# B&R Automation Studio project ACOPOStrak_DATech_Pilot (part 5)

#### actCodeReader.st
```iecst
ACTION actCodeReader:

	IF gSim THEN

		gInitialDone := TRUE;

	END_IF

	IF NOT gInitialDone THEN

	CASE CodeStep OF

		CODE_WAIT:

			IF gShuttleTotalCount > checkSHCount THEN

					fbTrig.Enable				:= TRUE;

				IF fbTrig.Valid THEN

					CodeStep				:= CODE_CHECK_TRIG;

				END_IF

			ELSE

				gInitialDone				:= TRUE;
				fbTrig.Enable				:= FALSE;
//				gBarCodeReader.Enable 		:= FALSE;

			END_IF

		CODE_CHECK_TRIG:

			IF fbTrig.EventCount > 0 THEN

				checkSHCount := checkSHCount + 1;

				fbTrigInfo.Execute := TRUE;

				fbUserData.DataAddress 			:= ADR(userData);
				fbUserData.DataSize 			:= SIZE_OF_USERDATA;
				fbUserData.Mode					:= mcACPTRAK_USERDATA_GET;
				fbUserData.Execute 				:= TRUE;

				CodeStep						:= CODE_GET_SH;

			END_IF

		CODE_GET_SH:

			IF fbTrigInfo.Done = TRUE AND fbUserData.Done = TRUE THEN

				Axis	:= fbTrigInfo.TrgPointInfo.Axis;
				fbUserData.Execute 				:= FALSE;

				CodeStep 				:= CODE_MOVE_TO_READER;

			END_IF

		CODE_MOVE_TO_READER:

			fbMovelAbs.Sector				:= ADR(SectorTrackAll);
			fbMovelAbs.Axis 				:= ADR(Axis);

			fbMovelAbs.Velocity				:= gPar.MovementPar.Initialize.Velocity;
			fbMovelAbs.Acceleration 		:= gPar.MovementPar.Initialize.Acceleration;
			fbMovelAbs.Deceleration 		:= gPar.MovementPar.Initialize.Deceleration;
			fbMovelAbs.Position				:= POS_VISION;

			fbMovelAbs.Execute 				:= TRUE;

			fbMovelAbs.AdvancedParameters.StartDirection 		:= mcDIR_UNDEFINED;
			fbMovelAbs.AdvancedParameters.EndDirection 			:= mcDIR_POSITIVE;

			fbMovelAbs.AdvancedParameters.ShuttleOrientation 	:= mcDIR_UNDEFINED;
			fbMovelAbs.AdvancedParameters.PosRelativeTo 		:= mcACPTRAK_SEC_START;

			IF fbMovelAbs.Done THEN

				fbMovelAbs.Execute 			:= FALSE;

				CodeStep					:= CODE_READER_CHECK;

			END_IF

		CODE_READER_CHECK:

			IF gVisionSensor.DAT.StatusText = 'Ready' AND NOT gVisionSensor.DAT.ImageProcessingActive THEN

				gBarCodeReader.Trigger		:= TRUE;
				checkTakeCount				:= gBarCodeReader.TakeCount;
				CodeStep					:= CODE_CHECK_TAKE_COUNT;

			END_IF

		CODE_CHECK_TAKE_COUNT:

			IF gVisionSensor.DAT.ImageProcessingActive AND checkTakeCount <> gBarCodeReader.TakeCount THEN // gVisionSensor.DAT.StatusText <> 'Ready' AND checkTakeCount <> gBarCodeReader.TakeCount THEN //bNextStep1 THEN

				gBarCodeReader.Trigger		:= FALSE;

				CodeStep					:= CODE_ID_DEFINE;

			END_IF

		CODE_ID_DEFINE:

			IF NOT gVisionSensor.DAT.ImageProcessingActive THEN // bNextStep2 THEN //

//				fbUserData.Axis 		:= ADR(Axis);
				fbUserData.Mode 		:= mcACPTRAK_USERDATA_SET;
				fbUserData.Execute 		:= TRUE;
				fbUserData.DataAddress	:= ADR(userData);
				fbUserData.DataSize		:= SIZEOF(userData);

//				StrShuttleCount 		:= USINT_TO_STRING(checkSHCount);
//
//				IF checkSHCount < 10 THEN
//					userData.SerialNumber		:= 'FA99999900';
//					userData.SerialNumber		:= CONCAT(userData.SerialNumber, StrShuttleCount);
//
//				ELSIF checkSHCount < 100 THEN
//					userData.SerialNumber		:= 'FA9999990';
//					userData.SerialNumber		:= CONCAT(userData.SerialNumber, StrShuttleCount);
//				END_IF

//				brsmemcpy(ADR(userData.SerialNumber), ADR(StrTempShuttleID), 11);// ADR(gBarCodeReader.SerialNumber), 11);

				userData.SerialNumber := gBarCodeReader.SerialNumber;

				IF fbUserData.Done = TRUE THEN // AND bNextStep3 THEN

					fbUserData.Execute 	:= FALSE;
					CodeStep					:= CODE_RELEASE_SH;

				END_IF

			END_IF

		CODE_RELEASE_SH:

			fbMovelVel.Sector				:= ADR(SectorTrackAll);
			fbMovelVel.Axis 				:= ADR(Axis);

			fbMovelVel.RouteVelocity 		:= gPar.MovementPar.Initialize.RoutedVelocity;
			fbMovelVel.Velocity 			:= gPar.MovementPar.Initialize.Velocity;
			fbMovelVel.Acceleration 		:= gPar.MovementPar.Initialize.Acceleration;
			fbMovelVel.Deceleration 		:= gPar.MovementPar.Initialize.Deceleration;

			fbMovelVel.Execute 				:= TRUE;

			fbMovelVel.AdvancedParameters.StartDirection 		:= mcDIR_UNDEFINED;
			fbMovelVel.AdvancedParameters.EndDirection 			:= mcDIR_POSITIVE;

			fbMovelVel.AdvancedParameters.ShuttleOrientation 	:= mcDIR_UNDEFINED;
			fbMovelVel.AdvancedParameters.PosRelativeTo 		:= mcACPTRAK_SEC_START;

			CodeStep 					:= CODE_NORMAL_END;

//			IF fbMovelVel.Active THEN
//
//				fbMovelVel.Execute 			:= FALSE;
//				fbUserData.Execute			:= FALSE;
//				fbTrigInfo.Execute			:= FALSE;
//
//			END_IF

		CODE_NORMAL_END:

			fbTrigInfo.Execute			:= FALSE;
			fbUserData.Execute			:= FALSE;
			fbMovelVel.Execute 			:= FALSE;

			CodeStep 					:= CODE_WAIT;

		END_CASE

	END_IF

	fbTrig();
	fbTrigInfo();
	fbUserData();
	fbMovelAbs();
	fbMovelVel();
	ShReadInfo();

	bMoveVelActive 	:= fbMovelVel.Active;

END_ACTION

ACTION actCodeReader_INIT:

	CodeStep 			:= CODE_WAIT;

//	gBarCodeReader.Enable 		:= FALSE;
//	gBarCodeReader.Trigger		:= FALSE;

	checkSHCount		:= 0;

	fbTrig.Enable		:= FALSE;
	fbTrigInfo.Execute	:= FALSE;
	fbUserData.Execute	:= FALSE;
	fbMovelAbs.Execute	:= FALSE;
	fbMovelVel.Execute	:= FALSE;

END_ACTION

/////////////////////////////////////////////////////////////////////////////////////////////////////////

//
//		INIT_BARRIERSETTING:(* Process Point Setting *)
//			countShuttle					:= 0;
//			gShuttleTotalCount				:= 0;
//
//			fbCheckInStatus.Enable 			:= TRUE;
//
//			fbCheckIn.Command 				:= mcACPTRAK_BARRIER_CLOSE;
//			fbCheckIn.Execute 				:= TRUE;
//
//			fbCheckOut.Command 				:= mcACPTRAK_BARRIER_OPEN;
//			fbCheckOut.Execute 				:= TRUE;
//
//			IF fbCheckIn.Done = TRUE AND fbCheckOut.Done = TRUE	AND fbCheckInStatus.Valid = TRUE THEN
//				fbCheckIn.Execute 			:= FALSE;
//				fbCheckOut.Execute 			:= FALSE;
//
//				fbAsmGetShuttle.Assembly 		:= ADR(gAsmMain);
//				fbAsmGetShuttle.Enable 			:= TRUE;
//
//				IF fbAsmGetShuttle.Valid = TRUE THEN
//					gShuttleTotalCount			:= fbAsmGetShuttle.TotalCount;
//					initStep 					:= INIT_SHUTTLE_CHECK;
//				END_IF
//			END_IF
//
//		INIT_SHUTTLE_CHECK:
//			IF fbAsmGetShuttle.TotalCount > countShuttle THEN
//				readShuttleInfo.Axis  		:= ADR(fbAsmGetShuttle.Axis);
//				readShuttleInfo.Enable 		:= TRUE;
//
//				IF readShuttleInfo.Valid = TRUE THEN
//					countShuttle			:= countShuttle + 1;
//					fbAsmGetShuttle.Next	:= FALSE;
//					initStep 				:= INIT_MOVE;
//				END_IF
//			ELSE
//				fbAsmGetShuttle.Enable 		:= FALSE;
//				readShuttleInfo.Enable 		:= FALSE;
//				initStep 					:= INIT_ADD_TICKET;
//			END_IF
//
//		INIT_MOVE:
//			IF readShuttleInfo.ShuttleInfo.CurrentValues.Velocity = 0 THEN
//				fbMovelVel.Sector				:= ADR(SecMain);
//				fbMovelVel.Axis 				:= ADR(fbAsmGetShuttle.Axis);
//
//				fbMovelVel.RouteVelocity 		:= gPar.MovementPar.Initialize.RoutedVelocity;
//				fbMovelVel.Velocity 			:= gPar.MovementPar.Initialize.Velocity;
//				fbMovelVel.Acceleration 		:= gPar.MovementPar.Initialize.Acceleration;
//				fbMovelVel.Deceleration 		:= gPar.MovementPar.Initialize.Deceleration;
//				fbMovelVel.Execute 				:= TRUE;
//
//				fbMovelVel.AdvancedParameters.StartDirection 		:= mcDIR_UNDEFINED;
//				fbMovelVel.AdvancedParameters.EndDirection 			:= mcDIR_POSITIVE;
//
//				fbMovelVel.AdvancedParameters.ShuttleOrientation 	:= mcDIR_UNDEFINED;
//				fbMovelVel.AdvancedParameters.PosRelativeTo 		:= mcACPTRAK_SEC_START;
//
//				IF bMoveVelActive = FALSE AND fbMovelVel.Active = TRUE THEN
//					fbMovelVel.Execute 			:= FALSE;
//					readShuttleInfo.Enable 		:= FALSE;
//					fbAsmGetShuttle.Next		:= TRUE;
//					initStep 					:= INIT_SHUTTLE_CHECK;
//				END_IF
//			END_IF
//
//		INIT_ADD_TICKET:
//			fbCheckIn.AdvancedParameters.TicketCount 	:= gShuttleTotalCount;
//			fbCheckIn.Command							:= mcACPTRAK_BARRIER_ADD_TICKETS;
//			fbCheckIn.Execute 							:= TRUE;
//
//			IF fbCheckIn.Done = TRUE THEN
//				fbCheckIn.Execute						:= FALSE;
//				initStep 								:= INIT_START_ID_IDENTIFICATION;
//			END_IF
//
//
//		INIT_START_ID_IDENTIFICATION:
//			IF fbCheckInStatus.BarrierInfo.RemainingTickets = 0 THEN
//				initStep 								:= INIT_CHECK_END;
//			END_IF
//
//		INIT_CHECK_END:
//			fbSecGetShuttles.Sector := ADR(SecMain);
//			fbSecGetShuttles.Enable := TRUE;
//			fbSecGetShuttles.AdvancedParameters.StartPosition 	:= 1.2;
//			fbSecGetShuttles.AdvancedParameters.EndPosition 	:= 2.4;
//
//			IF fbSecGetShuttles.Valid = TRUE THEN
//				IF fbSecGetShuttles.TotalCount = 0 THEN
//					fbSecGetShuttles.Enable 			:= FALSE;
//					initStep 							:= INIT_NORMAL_END;
//				ELSE
//					fbSecGetShuttles.Enable := FALSE;
//				END_IF
//			END_IF
//
//		INIT_NORMAL_END:
//			fbCheckInStatus.Enable := FALSE;
//			fbCheckIn.Execute := TRUE;
//			fbCheckOut.Execute := TRUE;
//
//			fbCheckIn.Command := mcACPTRAK_BARRIER_OPEN;
//			fbCheckOut.Command := mcACPTRAK_BARRIER_OPEN;
//
//			IF fbCheckIn.Done = TRUE AND fbCheckOut.Done = TRUE THEN
//				gSts.AsmState 					:= E_ASM_IDLE;
//			END_IF
//	END_CASE;
//
//	fbCheckInStatus();
//	fbCheckIn();
//	fbCheckOut();
//
//	fbAsmGetShuttle();
//	readShuttleInfo();
//
//	fbSecGetShuttles();
//
//	bMoveVelActive 	:= fbMovelVel.Active;
//
//END_ACTION
//
//ACTION actInitialize_INIT:
//	CodeStep 						:= CODE_WAIT;
//	fbAsmGetShuttle.Enable 			:= FALSE;
//	fbSecGetShuttles.Enable 		:= FALSE;
//	fbCheckInStatus.Enable			:= FALSE;
//	fbCheckIn.Execute 				:= FALSE;
//	fbCheckOut.Execute 				:= FALSE;
//	fbMovelVel.Execute				:= FALSE;
//END_ACTION
```

### Program Logical/Source/AsmControl/ctrCleanMode (IEC)

#### Variables.var
```iecst
VAR
	initStep : INT;
END_VAR
(**)
VAR
	fbSecGetShuttles : MC_BR_SecGetShuttleSel_AcpTrak;
END_VAR
(**)
VAR
	fbMovelVel : MC_BR_RoutedMoveVel_AcpTrak;
	fbMoveAbs : MC_BR_RoutedMoveAbs_AcpTrak;
END_VAR
(**)
VAR
	bMoveVelActive : BOOL;
END_VAR
(**)
VAR
	fbCheckOutStatus : MC_BR_BarrierReadInfo_AcpTrak;
	fbCheckInStatus : MC_BR_BarrierReadInfo_AcpTrak;
	fbCheckIn : MC_BR_BarrierCommand_AcpTrak;
	fbCheckOut : MC_BR_BarrierCommand_AcpTrak;
	fbCheckInTrg : MC_BR_TrgPointEnable_AcpTrak;
	fbCheckInTrgInfo : MC_BR_TrgPointGetInfo_AcpTrak;
	TotalShuttleCount : DINT;
END_VAR
```

#### Main.st
```iecst
PROGRAM _INIT

	fbCheckIn.ProcessPoint			:= ADR(ptCheckIn);
	fbCheckInStatus.ProcessPoint 	:= ADR(ptCheckIn);
	fbCheckInTrg.ProcessPoint		:= ADR(ptCheckIn);
	fbCheckInTrgInfo.ProcessPoint	:= ADR(ptCheckIn);

	fbCheckOutStatus.ProcessPoint	:= ADR(ptCheckOut);
	fbCheckOut.ProcessPoint			:= ADR(ptCheckOut);

END_PROGRAM

PROGRAM _CYCLIC

	IF gSts.AsmState <> E_ASM_CLEAN THEN
		initStep					:= 0;

		fbSecGetShuttles.Enable		:= FALSE;
		fbCheckInTrgInfo.Execute	:= FALSE;
		fbCheckIn.Execute			:= FALSE;
		fbCheckInStatus.Enable		:= FALSE;

		fbMoveAbs.Execute				:= FALSE;
		fbMovelVel.Execute 				:= FALSE;

		TotalShuttleCount				:= 0;
	ELSE

		CASE initStep OF
			0:
				fbCheckInStatus.Enable	:= TRUE;
				fbCheckIn.Execute 		:= TRUE;
				fbCheckOut.Execute 		:= TRUE;

				fbCheckIn.Command 		:= mcACPTRAK_BARRIER_OPEN;
				fbCheckOut.Command 		:= mcACPTRAK_BARRIER_OPEN;

				IF fbCheckIn.Done AND fbCheckInStatus.Valid THEN
					fbCheckIn.Execute 	:= FALSE;
					fbCheckOut.Execute 	:= FALSE;
					initStep			:= 10;
				END_IF

			10:
				fbSecGetShuttles.Sector := ADR(SectorTrackAll);
				fbSecGetShuttles.Enable := TRUE;
				fbSecGetShuttles.AdvancedParameters.StartPosition	:= 0.0;
				fbSecGetShuttles.AdvancedParameters.EndPosition		:= 0.0;

				IF fbSecGetShuttles.Valid = TRUE THEN
					TotalShuttleCount 	:= fbSecGetShuttles.TotalCount;
					initStep 			:= 20;
				END_IF

			20:
				fbSecGetShuttles.Next 			:= FALSE;

				fbMovelVel.Sector				:= ADR(SectorTrackAll);
				fbMovelVel.Axis 				:= ADR(fbSecGetShuttles.Axis);

				fbMovelVel.Position				:= 12.48;
				fbMovelVel.RouteVelocity 		:= 1.0;
				fbMovelVel.Velocity 			:= 1.0;
				fbMovelVel.Acceleration 		:= 1.0;
				fbMovelVel.Deceleration 		:= 1.0;
				fbMovelVel.Execute 				:= TRUE;

				fbMovelVel.AdvancedParameters.StartDirection 		:= mcDIR_POSITIVE;
				fbMovelVel.AdvancedParameters.EndDirection 			:= mcDIR_UNDEFINED;
				fbMovelVel.AdvancedParameters.ShuttleOrientation 	:= mcDIR_UNDEFINED;

				IF bMoveVelActive = FALSE AND fbMovelVel.Active = TRUE THEN
					fbMovelVel.Execute 			:= FALSE;
					initStep 					:= 30;
				END_IF

			30:
				IF fbSecGetShuttles.RemainingCount > 0 THEN
					fbSecGetShuttles.Next 		:= TRUE;
					initStep 					:= 20;
				ELSE
					fbSecGetShuttles.Enable 	:= FALSE;
			//		initStep 					:= 40;
				END_IF

			40:
				IF fbCheckInStatus.BarrierInfo.RemainingTickets = 0 THEN
					initStep 					:= 50;
				END_IF

			50:
				fbSecGetShuttles.Sector 		:= ADR(SectorTrackAll);
				fbSecGetShuttles.Enable 		:= TRUE;
				fbSecGetShuttles.AdvancedParameters.StartPosition 	:= 13.14;//12.48; // Check in point
				fbSecGetShuttles.AdvancedParameters.EndPosition 	:= 0.0;

				IF fbSecGetShuttles.Valid = TRUE AND fbSecGetShuttles.TotalCount = 0 THEN
					fbSecGetShuttles.Enable 		:= FALSE;
					initStep 						:= 60;
				ELSIF  fbSecGetShuttles.Valid = TRUE AND fbSecGetShuttles.TotalCount > 0 THEN
					fbSecGetShuttles.Enable 		:= FALSE;
				END_IF

			60:
				fbCheckInStatus.Enable := FALSE;
				fbCheckIn.Execute := TRUE;
				fbCheckOut.Execute := TRUE;

				fbCheckIn.Command := mcACPTRAK_BARRIER_OPEN;
				fbCheckOut.Command := mcACPTRAK_BARRIER_OPEN;

				IF fbCheckIn.Done = TRUE AND fbCheckOut.Done = TRUE THEN
					fbCheckIn.Execute 			:= FALSE;
					fbCheckOut.Execute 			:= FALSE;
					fbSecGetShuttles.Enable 	:= FALSE;
					gSts.AsmState 				:= E_ASM_IDLE;
					initStep 					:= 0;
				END_IF

		END_CASE;
	END_IF

	fbSecGetShuttles();

	fbCheckInTrg();
	fbCheckInTrgInfo();
	fbCheckIn();
	fbCheckInStatus();
	fbCheckOut();
	fbCheckOutStatus();
//	fbUserData();

	fbMoveAbs();
	bMoveVelActive 	:= fbMovelVel.Active;
	fbMovelVel();

END_PROGRAM

PROGRAM _EXIT
	(* Insert code here *)

END_PROGRAM
```

### Program Logical/Source/Control/ctrTransfer (IEC)

#### Main.st - Init, cyclic, exit code
```iecst
PROGRAM _INIT

	gSim	:= DiagCpuIsSimulated();

	StStage[0].Sector		:= ADR(SectorCurve1);
	StStage[1].Sector		:= ADR(SectorTrackA_2);
	StStage[2].Sector		:= ADR(SectorTrackA_2);
	StStage[3].Sector		:= ADR(SectorTrackA_2);
	StStage[4].Sector		:= ADR(SectorTrackA_2);
	StStage[5].Sector		:= ADR(SectorTrackA_2);
	StStage[6].Sector		:= ADR(SectorTrackA_2);
	StStage[7].Sector		:= ADR(SectorTrackA_2);
	StStage[8].Sector		:= ADR(SectorTrackA_2);
	StStage[9].Sector		:= ADR(SectorTrackA_3);
	StStage[10].Sector		:= ADR(SectorCurve3);
	StStage[11].Sector		:= ADR(SectorTrackA_4);
	StStage[12].Sector		:= ADR(SectorTrackA_4);
	StStage[13].Sector		:= ADR(SectorTrackA_4);
	StStage[14].Sector		:= ADR(SectorTrackA_4);
	StStage[15].Sector		:= ADR(SectorTrackA_4);
	StStage[16].Sector		:= ADR(SectorCurve4);
	StStage[17].Sector		:= ADR(SectorCurve4);
	StStage[18].Sector		:= ADR(SectorTrackA_1);

	/////////////////////////////////////////////////////////////////////////////////////
	// Can supply
	fbStage1.CheckInProcessPoint		:= ADR(ptCheckIn);
	fbStage1.CheckOutProcessPoint		:= ADR(ptCheckOut);
	fbStage1.TargetStage				:= ADR(StStage[0]);
	fbStage1.TargetSlotCount			:= COUNT_OF_SLOT;
	// TC insert
	fbStage2.SourceStage[0]				:= ADR(StStage[0]);
	fbStage2.SourceSlotCount[0]			:= COUNT_OF_SLOT;
	fbStage2.TargetStage				:= ADR(StStage[1]);
	fbStage2.TargetSlotCount			:= COUNT_OF_SLOT;
	// TC push
	fbStage3.SourceStage[0]				:= ADR(StStage[1]);
	fbStage3.SourceSlotCount[0]			:= COUNT_OF_SLOT;
	fbStage3.TargetStage				:= ADR(StStage[2]);
	fbStage3.TargetSlotCount			:= COUNT_OF_SLOT;
	// TC vision
	fbStage4.SourceStage[0]				:= ADR(StStage[2]);
	fbStage4.SourceSlotCount[0]			:= COUNT_OF_SLOT;
	fbStage4.TargetStage				:= ADR(StStage[3]);
	fbStage4.TargetSlotCount			:= COUNT_OF_SLOT;
	// TC NG re-insert
	fbStage5.SourceStage[0]				:= ADR(StStage[3]);
	fbStage5.SourceSlotCount[0]			:= COUNT_OF_SLOT;
	fbStage5.TargetStage				:= ADR(StStage[4]);
	fbStage5.TargetSlotCount			:= COUNT_OF_SLOT;
	// BCR vision
	fbStage6.SourceStage[0]				:= ADR(StStage[4]);
	fbStage6.SourceSlotCount[0]			:= COUNT_OF_SLOT;
	fbStage6.TargetStage				:= ADR(StStage[5]);
	fbStage6.TargetSlotCount			:= COUNT_OF_SLOT;
	// CCR 1
	fbStage7.SourceStage[0]				:= ADR(StStage[5]);
	fbStage7.SourceSlotCount[0]			:= COUNT_OF_SLOT;
	fbStage7.TargetStage				:= ADR(StStage[6]);
	fbStage7.TargetSlotCount			:= COUNT_OF_SLOT;
	// CCR 1 vision
	fbStage8.SourceStage[0]				:= ADR(StStage[6]);
	fbStage8.SourceSlotCount[0]			:= COUNT_OF_SLOT;
	fbStage8.TargetStage				:= ADR(StStage[7]);
	fbStage8.TargetSlotCount			:= COUNT_OF_SLOT;
	// CCR 2
	fbStage9.SourceStage[0]				:= ADR(StStage[7]);
	fbStage9.SourceSlotCount[0]			:= COUNT_OF_SLOT;
	fbStage9.TargetStage				:= ADR(StStage[8]);
	fbStage9.TargetSlotCount			:= COUNT_OF_SLOT;
	// Maint
	fbStage10.SourceStage[0]			:= ADR(StStage[8]);
	fbStage10.SourceSlotCount[0]		:= COUNT_OF_SLOT;
	fbStage10.TargetStage				:= ADR(StStage[9]);
	fbStage10.TargetSlotCount			:= COUNT_OF_SLOT;
	// CCR 2 vision
	fbStage11.SourceStage[0]			:= ADR(StStage[9]);
	fbStage11.SourceSlotCount[0]		:= COUNT_OF_SLOT;
	fbStage11.TargetStage				:= ADR(StStage[10]);
	fbStage11.TargetSlotCount			:= COUNT_OF_SLOT;
	// CCR 3
	fbStage12.SourceStage[0]			:= ADR(StStage[10]);
	fbStage12.SourceSlotCount[0]		:= COUNT_OF_SLOT;
	fbStage12.TargetStage				:= ADR(StStage[11]);
	fbStage12.TargetSlotCount			:= COUNT_OF_SLOT;
	// CCR 3 vision
	fbStage13.SourceStage[0]			:= ADR(StStage[11]);
	fbStage13.SourceSlotCount[0]		:= COUNT_OF_SLOT;
	fbStage13.TargetStage				:= ADR(StStage[12]);
	fbStage13.TargetSlotCount			:= COUNT_OF_SLOT;
	// CSZ
	fbStage14.SourceStage[0]			:= ADR(StStage[12]);
	fbStage14.SourceSlotCount[0]		:= COUNT_OF_SLOT;
	fbStage14.TargetStage				:= ADR(StStage[13]);
	fbStage14.TargetSlotCount			:= COUNT_OF_SLOT;
	// 3D done position
	fbStage15.SourceStage[0]			:= ADR(StStage[13]);
	fbStage15.SourceSlotCount[0]		:= COUNT_OF_SLOT;
	fbStage15.TargetStage				:= ADR(StStage[14]);
	fbStage15.TargetSlotCount			:= COUNT_OF_SLOT;
	// Diameter inspection
	fbStage16.SourceStage[0]			:= ADR(StStage[14]);
	fbStage16.SourceSlotCount[0]		:= COUNT_OF_SLOT;
	fbStage16.TargetStage				:= ADR(StStage[15]);
	fbStage16.TargetSlotCount			:= COUNT_OF_SLOT;
	// NG out
	fbStage17.SourceStage[0]			:= ADR(StStage[15]);
	fbStage17.SourceSlotCount[0]		:= COUNT_OF_SLOT;
	fbStage17.TargetStage				:= ADR(StStage[16]);
	fbStage17.TargetSlotCount			:= COUNT_OF_SLOT;
	// Unloading
	fbStage18.SourceStage[0]			:= ADR(StStage[16]);
	fbStage18.SourceSlotCount[0]		:= COUNT_OF_SLOT;
	fbStage18.TargetStage				:= ADR(StStage[17]);
	fbStage18.TargetSlotCount			:= COUNT_OF_SLOT;
	// Clean
	fbStage19.SourceStage[0]			:= ADR(StStage[17]);
	fbStage19.SourceSlotCount[0]		:= COUNT_OF_SLOT;
	fbStage19.TargetStage				:= ADR(StStage[18]);
	fbStage19.TargetSlotCount			:= COUNT_OF_SLOT;
	// Return
	fbReturn.SourceStage[0]				:= ADR(StStage[18]);
	fbReturn.SourceSlotCount[0]			:= COUNT_OF_SLOT;
	fbReturn.TargetSector				:= ADR(SectorTrackAll);
	fbReturn.TargetPosition				:= 12.5;
	/////////////////////////////////////////////////////////////////////////////////////
	InitializeFcBank(30);

	actParameterInitialize;

	/////////////////////////////////////////////////////////////////////////////////////
	// Buffer
	/////////////////////////////////////////////////////////////////////////////////////

	//Wait buffer for CSZ
	fbCSZWait.InPoint				:= ADR(ptCSZIn);
	fbCSZWait.OutPoint				:= ADR(ptCSZOut);
	fbCSZWait.MaximumShuttleCount	:= 1;
	//fbCSZWait.InitShuttleCount		:= 1;

	//Wait for unloading
	fbUnloadingWait.InPoint				:= ADR(ptUnloadingIn);
	fbUnloadingWait.OutPoint			:= ADR(ptUnloadingOut);
	fbUnloadingWait.MaximumShuttleCount	:= 1;
	fbUnloadingWait.InitShuttleCount	:= 1;

END_PROGRAM

PROGRAM _CYCLIC

	actUpdateParamter;

	CASE gSts.AsmState OF
		E_ASM_INITIALIZATION:
			//For Initialize Slot Status.
			FOR i := 0 TO 18 DO
				StStage[i].Interface	:= E_SLOT_UNKNOWN;
			END_FOR;

		E_ASM_MANUAL:

			fbStage1(Enable := TRUE, Process := FALSE, Feeding := FALSE);
			fbStage2(Enable := TRUE, Process := FALSE);
			fbStage3(Enable := TRUE, Process := FALSE);
			fbStage4(Enable := TRUE, Process := FALSE);
			fbStage5(Enable := TRUE, Process := FALSE);
			fbStage6(Enable := TRUE, Process := FALSE);
			fbStage7(Enable := TRUE, Process := FALSE);
			fbStage8(Enable := TRUE, Process := FALSE);
			fbStage9(Enable := TRUE, Process := FALSE);
			fbStage10(Enable := TRUE, Process := FALSE);
			fbStage11(Enable := TRUE, Process := FALSE);
			fbStage12(Enable := TRUE, Process := FALSE);
			fbStage13(Enable := TRUE, Process := FALSE);
			fbStage14(Enable := TRUE, Process := FALSE);
			fbStage15(Enable := TRUE, Process := FALSE);
			fbStage16(Enable := TRUE, Process := FALSE);
			fbStage17(Enable := TRUE, Process := FALSE);
			fbStage18(Enable := TRUE, Process := FALSE);
			fbStage19(Enable := TRUE, Process := FALSE);
			fbReturn(Enable := TRUE, Process := FALSE);
			fbCSZWait(Enable := FALSE);
			fbUnloadingWait(Enable := FALSE);

			FOR i := 0 TO 18 DO
				StStage[i].Interface	:= E_SLOT_MANUAL;

				IF i < 18 THEN
					StStage[i].NextStage	:= ADR(StStage[i + 1]);
				ELSIF i = 18 THEN
					StStage[18].NextStage	:= ADR(StStage[0]);
				END_IF
			END_FOR;

		E_ASM_IDLE:

			fbStage1(Enable := TRUE, Process := TRUE, Feeding := FALSE);
			fbStage2(Enable := TRUE, Process := TRUE);
			fbStage3(Enable := TRUE, Process := TRUE);
			fbStage4(Enable := TRUE, Process := TRUE);
			fbStage5(Enable := TRUE, Process := TRUE);
			fbStage6(Enable := TRUE, Process := TRUE);
			fbStage7(Enable := TRUE, Process := TRUE);
			fbStage8(Enable := TRUE, Process := TRUE);
			fbStage9(Enable := TRUE, Process := TRUE);
			fbStage10(Enable := TRUE, Process := TRUE);
			fbStage11(Enable := TRUE, Process := TRUE);
			fbStage12(Enable := TRUE, Process := TRUE);
			fbStage13(Enable := TRUE, Process := TRUE);
			fbStage14(Enable := TRUE, Process := TRUE);
			fbStage15(Enable := TRUE, Process := TRUE);
			fbStage16(Enable := TRUE, Process := TRUE);
			fbStage17(Enable := TRUE, Process := TRUE);
			fbStage18(Enable := TRUE, Process := TRUE);
			fbStage19(Enable := TRUE, Process := TRUE);
			fbReturn(Enable := TRUE, Process := TRUE);
			fbCSZWait(Enable := TRUE);
			fbUnloadingWait(Enable := TRUE);

		E_ASM_PROCESS:

			fbStage1(Enable := TRUE, Process := TRUE, Feeding := TRUE);
			fbStage2(Enable := TRUE, Process := TRUE);
			fbStage3(Enable := TRUE, Process := TRUE);
			fbStage4(Enable := TRUE, Process := TRUE);
			fbStage5(Enable := TRUE, Process := TRUE);
			fbStage6(Enable := TRUE, Process := TRUE);
			fbStage7(Enable := TRUE, Process := TRUE);
			fbStage8(Enable := TRUE, Process := TRUE);
			fbStage9(Enable := TRUE, Process := TRUE);
			fbStage10(Enable := TRUE, Process := TRUE);
			fbStage11(Enable := TRUE, Process := TRUE);
			fbStage12(Enable := TRUE, Process := TRUE);
			fbStage13(Enable := TRUE, Process := TRUE);
			fbStage14(Enable := TRUE, Process := TRUE);
			fbStage15(Enable := TRUE, Process := TRUE);
			fbStage16(Enable := TRUE, Process := TRUE);
			fbStage17(Enable := TRUE, Process := TRUE);
			fbStage18(Enable := TRUE, Process := TRUE);
			fbStage19(Enable := TRUE, Process := TRUE);
			fbReturn(Enable := TRUE, Process := TRUE);
			fbCSZWait(Enable := TRUE);
			fbUnloadingWait(Enable := TRUE);

		E_ASM_STOPPING:

			fbStage1(Enable := TRUE, Process := TRUE, Feeding := FALSE);
			fbStage2(Enable := TRUE, Process := TRUE);
			fbStage3(Enable := TRUE, Process := TRUE);
			fbStage4(Enable := TRUE, Process := TRUE);
			fbStage5(Enable := TRUE, Process := TRUE);
			fbStage6(Enable := TRUE, Process := TRUE);
			fbStage7(Enable := TRUE, Process := TRUE);
			fbStage8(Enable := TRUE, Process := TRUE);
			fbStage9(Enable := TRUE, Process := TRUE);
			fbStage10(Enable := TRUE, Process := TRUE);
			fbStage11(Enable := TRUE, Process := TRUE);
			fbStage12(Enable := TRUE, Process := TRUE);
			fbStage13(Enable := TRUE, Process := TRUE);
			fbStage14(Enable := TRUE, Process := TRUE);
			fbStage15(Enable := TRUE, Process := TRUE);
			fbStage16(Enable := TRUE, Process := TRUE);
			fbStage17(Enable := TRUE, Process := TRUE);
			fbStage18(Enable := TRUE, Process := TRUE);
			fbStage19(Enable := TRUE, Process := TRUE);
			fbReturn(Enable := TRUE, Process := TRUE);
			fbCSZWait(Enable := TRUE);
			fbUnloadingWait(Enable := TRUE);

			IF fbStage1.ErrorID = MyTrakIdle AND
				fbStage2.ErrorID = MyTrakIdle AND
				fbStage3.ErrorID = MyTrakIdle AND
				fbStage4.ErrorID = MyTrakIdle AND
				fbStage5.ErrorID = MyTrakIdle AND
				fbStage6.ErrorID = MyTrakIdle AND
				fbStage7.ErrorID = MyTrakIdle AND
				fbStage8.ErrorID = MyTrakIdle AND
				fbStage9.ErrorID = MyTrakIdle AND
				fbStage10.ErrorID = MyTrakIdle AND
				fbStage11.ErrorID = MyTrakIdle AND
				fbStage12.ErrorID = MyTrakIdle AND
				fbStage13.ErrorID = MyTrakIdle AND
				fbStage14.ErrorID = MyTrakIdle AND
				fbStage15.ErrorID = MyTrakIdle AND
				fbStage16.ErrorID = MyTrakIdle AND
				fbStage17.ErrorID = MyTrakIdle AND
				fbStage18.ErrorID = MyTrakIdle AND
				fbStage19.ErrorID = MyTrakIdle AND

				StStage[0].Interface = E_SLOT_IDLE AND
				StStage[1].Interface = E_SLOT_IDLE AND
				StStage[2].Interface = E_SLOT_IDLE AND
				StStage[3].Interface = E_SLOT_IDLE AND
				StStage[4].Interface = E_SLOT_IDLE AND
				StStage[5].Interface = E_SLOT_IDLE AND
				StStage[6].Interface = E_SLOT_IDLE AND
				StStage[7].Interface = E_SLOT_IDLE AND
				StStage[8].Interface = E_SLOT_IDLE AND
				StStage[9].Interface = E_SLOT_IDLE AND
				StStage[10].Interface = E_SLOT_IDLE AND
				StStage[11].Interface = E_SLOT_IDLE AND
				StStage[12].Interface = E_SLOT_IDLE AND
				StStage[13].Interface = E_SLOT_IDLE AND
				StStage[14].Interface = E_SLOT_IDLE AND
				StStage[15].Interface = E_SLOT_IDLE AND
				StStage[16].Interface = E_SLOT_IDLE AND
				StStage[17].Interface = E_SLOT_IDLE AND
				StStage[18].Interface = E_SLOT_IDLE	THEN
			//	gSts.AsmState	:= E_ASM_IDLE;
			END_IF

		ELSE
			fbStage1(Enable := FALSE, Process := FALSE, Feeding := FALSE);
			fbStage2(Enable := FALSE, Process := FALSE);
			fbStage3(Enable := FALSE, Process := FALSE);
			fbStage4(Enable := FALSE, Process := FALSE);
			fbStage5(Enable := FALSE, Process := FALSE);
			fbStage6(Enable := FALSE, Process := FALSE);
			fbStage7(Enable := FALSE, Process := FALSE);
			fbStage8(Enable := FALSE, Process := FALSE);
			fbStage9(Enable := FALSE, Process := FALSE);
			fbStage10(Enable := FALSE, Process := FALSE);
			fbStage11(Enable := FALSE, Process := FALSE);
			fbStage12(Enable := FALSE, Process := FALSE);
			fbStage13(Enable := FALSE, Process := FALSE);
			fbStage14(Enable := FALSE, Process := FALSE);
			fbStage15(Enable := FALSE, Process := FALSE);
			fbStage16(Enable := FALSE, Process := FALSE);
			fbStage17(Enable := FALSE, Process := FALSE);
			fbStage18(Enable := FALSE, Process := FALSE);
			fbStage19(Enable := FALSE, Process := FALSE);
			fbReturn(Enable := FALSE, Process := FALSE);
			fbCSZWait(Enable := FALSE);
			fbUnloadingWait(Enable := FALSE);

	END_CASE;

	readShuttleInfo.Axis	:= ADR(StStage[0].Shuttle);
	readShuttleInfo();

END_PROGRAM

PROGRAM _EXIT

	fbStage1.Enable		:= FALSE;
	fbStage2.Enable		:= FALSE;
	fbStage3.Enable		:= FALSE;
	fbStage4.Enable		:= FALSE;
	fbStage5.Enable		:= FALSE;
	fbStage6.Enable		:= FALSE;
	fbStage7.Enable		:= FALSE;
	fbStage8.Enable		:= FALSE;
	fbStage9.Enable		:= FALSE;
	fbStage10.Enable	:= FALSE;
	fbStage11.Enable	:= FALSE;
	fbStage12.Enable	:= FALSE;
	fbStage13.Enable	:= FALSE;
	fbStage14.Enable	:= FALSE;
	fbStage15.Enable	:= FALSE;
	fbStage16.Enable	:= FALSE;
	fbStage17.Enable	:= FALSE;
	fbStage18.Enable	:= FALSE;
	fbStage19.Enable	:= FALSE;
	fbCSZWait.Enable	:= FALSE;

END_PROGRAM
```

#### Variables.var - Local variables
```iecst
VAR
	fbStage1 : MyTrak_Buffer; (*can supply*)
	fbStage2 : MyTrak_TransStage; (*TC insert*)
	fbStage3 : MyTrak_TransStage; (*TC push*)
	fbStage4 : MyTrak_TransStage; (*TC vision*)
	fbStage5 : MyTrak_TransStage; (*TC NG re-insert*)
	fbStage6 : MyTrak_TransStage; (*BCR vision*)
	fbStage7 : MyTrak_TransStage; (*CCR 1*)
	fbStage8 : MyTrak_TransStage; (*CCR 1 vision*)
	fbStage9 : MyTrak_TransStage; (*CCR 2 *)
	fbStage10 : MyTrak_TransStage; (*Maint*)
	fbStage11 : MyTrak_TransStage; (*CCR 2 vision*)
	fbStage12 : MyTrak_TransStage; (*CCR 3*)
	fbStage13 : MyTrak_TransStage; (*CCR 3 vision*)
	fbStage14 : MyTrak_TransStage; (*CSZ*)
	fbStage15 : MyTrak_TransStage; (*3D scan done position*)
	fbStage16 : MyTrak_TransStage; (*Diameter inspection*)
	fbStage17 : MyTrak_TransStage; (*NG out*)
	fbStage18 : MyTrak_TransStage; (*unloading*)
	fbStage19 : MyTrak_TransStage; (*Clean*)
	fbReturn : MyTrak_Serialize;
	fbCSZWait : MyTrak_TicketArea;
	fbUnloadingWait : MyTrak_TicketArea;
END_VAR
(**)
VAR
	readShuttleInfo : MC_BR_ShReadInfo_AcpTrak;
	i : USINT;
END_VAR
```

#### actUpdateParameter.st
```iecst
ACTION actUpdateParamter:

	// Stage pararmeter setting
	FOR i := 0 TO 18 DO
		StStage[i].Enable	:= TRUE;
	END_FOR;

	StStage[0].Position			:= POS_STAGE1 + gPar.PositionOffset.Stage[0];
	StStage[1].Position			:= POS_STAGE2 + gPar.PositionOffset.Stage[1];
	StStage[2].Position			:= POS_STAGE3 + gPar.PositionOffset.Stage[2];
	StStage[3].Position			:= POS_STAGE4 + gPar.PositionOffset.Stage[3];
	StStage[4].Position			:= POS_STAGE5 + gPar.PositionOffset.Stage[4];
	StStage[5].Position			:= POS_STAGE6 + gPar.PositionOffset.Stage[5];
	StStage[6].Position			:= POS_STAGE7 + gPar.PositionOffset.Stage[6];
	StStage[7].Position			:= POS_STAGE8 + gPar.PositionOffset.Stage[7];
	StStage[8].Position			:= POS_STAGE9 + gPar.PositionOffset.Stage[8];
	StStage[9].Position			:= POS_STAGE10 + gPar.PositionOffset.Stage[9];
	StStage[10].Position		:= POS_STAGE11 + gPar.PositionOffset.Stage[10];
	StStage[11].Position		:= POS_STAGE12 + gPar.PositionOffset.Stage[11];
	StStage[12].Position		:= POS_STAGE13 + gPar.PositionOffset.Stage[12];
	StStage[13].Position		:= POS_STAGE14 + gPar.PositionOffset.Stage[13];
	StStage[14].Position		:= POS_STAGE15 + gPar.PositionOffset.Stage[14];
	StStage[15].Position		:= POS_STAGE16 + gPar.PositionOffset.Stage[15];
	StStage[16].Position		:= POS_STAGE17 + gPar.PositionOffset.Stage[16];
	StStage[17].Position		:= POS_STAGE18 + gPar.PositionOffset.Stage[17];
	StStage[18].Position		:= POS_STAGE19 + gPar.PositionOffset.Stage[18];

	// Movement pararmeter setting

	fbStage1.SetPPM										:= gPar.TargetPPM;
	fbStage1.CountOfOneShot								:= gPar.CountOfGroup;
	fbStage1.Velocity									:= gPar.MovementPar.Stage1.Velocity;
	fbStage1.Acceleration								:= gPar.MovementPar.Stage1.Acceleration;
	fbStage1.Deceleration								:= gPar.MovementPar.Stage1.Deceleration;
	fbStage1.AdvancedParameters.StartDirection 			:= mcDIR_POSITIVE;
	fbStage1.AdvancedParameters.EndDirection 			:= mcDIR_UNDEFINED;
	fbStage1.AdvancedParameters.ShuttleOrientation 		:= mcDIR_UNDEFINED;
	fbStage1.MaximumShuttleCount						:= gPar.MovementPar.Stage1.MaxController;

	fbStage2.Velocity									:= gPar.MovementPar.Stage2.Velocity;
	fbStage2.Acceleration								:= gPar.MovementPar.Stage2.Acceleration;
	fbStage2.Deceleration								:= gPar.MovementPar.Stage2.Deceleration;
	fbStage2.AdvancedParameters.StartDirection 			:= mcDIR_POSITIVE;
	fbStage2.AdvancedParameters.EndDirection 			:= mcDIR_UNDEFINED;
	fbStage2.AdvancedParameters.ShuttleOrientation 		:= mcDIR_UNDEFINED;
	fbStage2.MaximumShuttleCount						:= gPar.MovementPar.Stage2.MaxController;

	fbStage3.Velocity									:= gPar.MovementPar.Stage3.Velocity;
	fbStage3.Acceleration								:= gPar.MovementPar.Stage3.Acceleration;
	fbStage3.Deceleration								:= gPar.MovementPar.Stage3.Deceleration;
	fbStage3.AdvancedParameters.StartDirection 			:= mcDIR_POSITIVE;
	fbStage3.AdvancedParameters.EndDirection 			:= mcDIR_UNDEFINED;
	fbStage3.AdvancedParameters.ShuttleOrientation 		:= mcDIR_UNDEFINED;
	fbStage3.MaximumShuttleCount						:= gPar.MovementPar.Stage3.MaxController;

	fbStage4.Velocity									:= gPar.MovementPar.Stage4.Velocity;
	fbStage4.Acceleration								:= gPar.MovementPar.Stage4.Acceleration;
	fbStage4.Deceleration								:= gPar.MovementPar.Stage4.Deceleration;
	fbStage4.AdvancedParameters.StartDirection 			:= mcDIR_POSITIVE;
	fbStage4.AdvancedParameters.EndDirection 			:= mcDIR_UNDEFINED;
	fbStage4.AdvancedParameters.ShuttleOrientation 		:= mcDIR_UNDEFINED;
	fbStage4.MaximumShuttleCount						:= gPar.MovementPar.Stage4.MaxController;

	fbStage5.Velocity									:= gPar.MovementPar.Stage5.Velocity;
	fbStage5.Acceleration								:= gPar.MovementPar.Stage5.Acceleration;
	fbStage5.Deceleration								:= gPar.MovementPar.Stage5.Deceleration;
	fbStage5.AdvancedParameters.StartDirection 			:= mcDIR_POSITIVE;
	fbStage5.AdvancedParameters.EndDirection 			:= mcDIR_UNDEFINED;
	fbStage5.AdvancedParameters.ShuttleOrientation 		:= mcDIR_UNDEFINED;
	fbStage5.MaximumShuttleCount						:= gPar.MovementPar.Stage5.MaxController;

	fbStage6.Velocity									:= gPar.MovementPar.Stage6.Velocity;
	fbStage6.Acceleration								:= gPar.MovementPar.Stage6.Acceleration;
	fbStage6.Deceleration								:= gPar.MovementPar.Stage6.Deceleration;
	fbStage6.AdvancedParameters.StartDirection 			:= mcDIR_POSITIVE;
	fbStage6.AdvancedParameters.EndDirection 			:= mcDIR_UNDEFINED;
	fbStage6.AdvancedParameters.ShuttleOrientation 		:= mcDIR_UNDEFINED;
	fbStage6.MaximumShuttleCount						:= gPar.MovementPar.Stage6.MaxController;

	fbStage7.Velocity									:= gPar.MovementPar.Stage7.Velocity;
	fbStage7.Acceleration								:= gPar.MovementPar.Stage7.Acceleration;
	fbStage7.Deceleration								:= gPar.MovementPar.Stage7.Deceleration;
	fbStage7.AdvancedParameters.StartDirection 			:= mcDIR_POSITIVE;
	fbStage7.AdvancedParameters.EndDirection 			:= mcDIR_UNDEFINED;
	fbStage7.AdvancedParameters.ShuttleOrientation 		:= mcDIR_UNDEFINED;
	fbStage7.MaximumShuttleCount						:= gPar.MovementPar.Stage7.MaxController;

	fbStage8.Velocity									:= gPar.MovementPar.Stage8.Velocity;
	fbStage8.Acceleration								:= gPar.MovementPar.Stage8.Acceleration;
	fbStage8.Deceleration								:= gPar.MovementPar.Stage8.Deceleration;
	fbStage8.AdvancedParameters.StartDirection 			:= mcDIR_POSITIVE;
	fbStage8.AdvancedParameters.EndDirection 			:= mcDIR_UNDEFINED;
	fbStage8.AdvancedParameters.ShuttleOrientation 		:= mcDIR_UNDEFINED;
	fbStage8.MaximumShuttleCount						:= gPar.MovementPar.Stage8.MaxController;

	fbStage9.Velocity									:= gPar.MovementPar.Stage9.Velocity;
	fbStage9.Acceleration								:= gPar.MovementPar.Stage9.Acceleration;
	fbStage9.Deceleration								:= gPar.MovementPar.Stage9.Deceleration;
	fbStage9.AdvancedParameters.StartDirection 			:= mcDIR_POSITIVE;
	fbStage9.AdvancedParameters.EndDirection 			:= mcDIR_UNDEFINED;
	fbStage9.AdvancedParameters.ShuttleOrientation 		:= mcDIR_UNDEFINED;
	fbStage9.MaximumShuttleCount						:= gPar.MovementPar.Stage9.MaxController;

	fbStage10.Velocity									:= gPar.MovementPar.Stage10.Velocity;
	fbStage10.Acceleration								:= gPar.MovementPar.Stage10.Acceleration;
	fbStage10.Deceleration								:= gPar.MovementPar.Stage10.Deceleration;
	fbStage10.AdvancedParameters.StartDirection 		:= mcDIR_POSITIVE;
	fbStage10.AdvancedParameters.EndDirection 			:= mcDIR_UNDEFINED;
	fbStage10.AdvancedParameters.ShuttleOrientation 	:= mcDIR_UNDEFINED;
	fbStage10.MaximumShuttleCount						:= gPar.MovementPar.Stage10.MaxController;

	fbStage11.Velocity									:= gPar.MovementPar.Stage11.Velocity;
	fbStage11.Acceleration								:= gPar.MovementPar.Stage11.Acceleration;
	fbStage11.Deceleration								:= gPar.MovementPar.Stage11.Deceleration;
	fbStage11.AdvancedParameters.StartDirection 		:= mcDIR_POSITIVE;
	fbStage11.AdvancedParameters.EndDirection 			:= mcDIR_UNDEFINED;
	fbStage11.AdvancedParameters.ShuttleOrientation 	:= mcDIR_UNDEFINED;
	fbStage11.MaximumShuttleCount						:= gPar.MovementPar.Stage11.MaxController;

	fbStage12.Velocity									:= gPar.MovementPar.Stage12.Velocity;
	fbStage12.Acceleration								:= gPar.MovementPar.Stage12.Acceleration;
	fbStage12.Deceleration								:= gPar.MovementPar.Stage12.Deceleration;
	fbStage12.AdvancedParameters.StartDirection 		:= mcDIR_POSITIVE;
	fbStage12.AdvancedParameters.EndDirection 			:= mcDIR_UNDEFINED;
	fbStage12.AdvancedParameters.ShuttleOrientation 	:= mcDIR_UNDEFINED;
	fbStage12.MaximumShuttleCount						:= gPar.MovementPar.Stage12.MaxController;

	fbStage13.Velocity									:= gPar.MovementPar.Stage13.Velocity;
	fbStage13.Acceleration								:= gPar.MovementPar.Stage13.Acceleration;
	fbStage13.Deceleration								:= gPar.MovementPar.Stage13.Deceleration;
	fbStage13.AdvancedParameters.StartDirection 		:= mcDIR_POSITIVE;
	fbStage13.AdvancedParameters.EndDirection 			:= mcDIR_UNDEFINED;
	fbStage13.AdvancedParameters.ShuttleOrientation 	:= mcDIR_UNDEFINED;
	fbStage13.MaximumShuttleCount						:= gPar.MovementPar.Stage13.MaxController;

	fbStage14.Velocity									:= gPar.MovementPar.Stage14.Velocity;
	fbStage14.Acceleration								:= gPar.MovementPar.Stage14.Acceleration;
	fbStage14.Deceleration								:= gPar.MovementPar.Stage14.Deceleration;
	fbStage14.AdvancedParameters.StartDirection 		:= mcDIR_POSITIVE;
	fbStage14.AdvancedParameters.EndDirection 			:= mcDIR_UNDEFINED;
	fbStage14.AdvancedParameters.ShuttleOrientation 	:= mcDIR_UNDEFINED;
	fbStage14.MaximumShuttleCount						:= gPar.MovementPar.Stage14.MaxController;

	fbStage15.Velocity									:= gPar.MovementPar.Stage15.Velocity;
	fbStage15.Acceleration								:= gPar.MovementPar.Stage15.Acceleration;
	fbStage15.Deceleration								:= gPar.MovementPar.Stage15.Deceleration;
	fbStage15.AdvancedParameters.StartDirection 		:= mcDIR_POSITIVE;
	fbStage15.AdvancedParameters.EndDirection 			:= mcDIR_UNDEFINED;
	fbStage15.AdvancedParameters.ShuttleOrientation 	:= mcDIR_UNDEFINED;
	fbStage15.MaximumShuttleCount						:= gPar.MovementPar.Stage15.MaxController;

	fbStage16.Velocity									:= gPar.MovementPar.Stage16.Velocity;
	fbStage16.Acceleration								:= gPar.MovementPar.Stage16.Acceleration;
	fbStage16.Deceleration								:= gPar.MovementPar.Stage16.Deceleration;
	fbStage16.AdvancedParameters.StartDirection 		:= mcDIR_POSITIVE;
	fbStage16.AdvancedParameters.EndDirection 			:= mcDIR_UNDEFINED;
	fbStage16.AdvancedParameters.ShuttleOrientation 	:= mcDIR_UNDEFINED;
	fbStage16.MaximumShuttleCount						:= gPar.MovementPar.Stage16.MaxController;

	fbStage17.Velocity									:= gPar.MovementPar.Stage17.Velocity;
	fbStage17.Acceleration								:= gPar.MovementPar.Stage17.Acceleration;
	fbStage17.Deceleration								:= gPar.MovementPar.Stage17.Deceleration;
	fbStage17.AdvancedParameters.StartDirection 		:= mcDIR_POSITIVE;
	fbStage17.AdvancedParameters.EndDirection 			:= mcDIR_UNDEFINED;
	fbStage17.AdvancedParameters.ShuttleOrientation 	:= mcDIR_UNDEFINED;
	fbStage17.MaximumShuttleCount						:= gPar.MovementPar.Stage17.MaxController;

	fbStage18.Velocity									:= gPar.MovementPar.Stage18.Velocity;
	fbStage18.Acceleration								:= gPar.MovementPar.Stage18.Acceleration;
	fbStage18.Deceleration								:= gPar.MovementPar.Stage18.Deceleration;
	fbStage18.AdvancedParameters.StartDirection 		:= mcDIR_POSITIVE;
	fbStage18.AdvancedParameters.EndDirection 			:= mcDIR_UNDEFINED;
	fbStage18.AdvancedParameters.ShuttleOrientation 	:= mcDIR_UNDEFINED;
	fbStage18.MaximumShuttleCount						:= gPar.MovementPar.Stage18.MaxController;

	fbStage19.Velocity									:= gPar.MovementPar.Stage19.Velocity;
	fbStage19.Acceleration								:= gPar.MovementPar.Stage19.Acceleration;
	fbStage19.Deceleration								:= gPar.MovementPar.Stage19.Deceleration;
	fbStage19.AdvancedParameters.StartDirection 		:= mcDIR_POSITIVE;
	fbStage19.AdvancedParameters.EndDirection 			:= mcDIR_UNDEFINED;
	fbStage19.AdvancedParameters.ShuttleOrientation 	:= mcDIR_UNDEFINED;
	fbStage19.MaximumShuttleCount						:= gPar.MovementPar.Stage19.MaxController;

	fbReturn.RoutedVelocity								:= gPar.MovementPar.Return.RoutedVelocity;
	fbReturn.Velocity									:= gPar.MovementPar.Return.Velocity;
	fbReturn.Acceleration								:= gPar.MovementPar.Return.Acceleration;
	fbReturn.Deceleration								:= gPar.MovementPar.Return.Deceleration;
	fbReturn.AdvancedParameters.StartDirection 			:= mcDIR_POSITIVE;
	fbReturn.AdvancedParameters.EndDirection 			:= mcDIR_UNDEFINED;
	fbReturn.AdvancedParameters.ShuttleOrientation		:= mcDIR_UNDEFINED;

END_ACTION
```

#### actParameterInitialize.st
```iecst
ACTION actParameterInitialize:
	IF gParInitialized = FALSE THEN
		// Position Parameter Intialize
		gPar.ProcessPosition.Stage[0]						:= POS_STAGE1;
		gPar.ProcessPosition.Stage[1]						:= POS_STAGE2;
		gPar.ProcessPosition.Stage[2]						:= POS_STAGE3;
		gPar.ProcessPosition.Stage[3]						:= POS_STAGE4;
		gPar.ProcessPosition.Stage[4]						:= POS_STAGE5;
		gPar.ProcessPosition.Stage[5]						:= POS_STAGE6;
		gPar.ProcessPosition.Stage[6]						:= POS_STAGE7;
		gPar.ProcessPosition.Stage[7]						:= POS_STAGE8;
		gPar.ProcessPosition.Stage[8]						:= POS_STAGE9;
		gPar.ProcessPosition.Stage[9]						:= POS_STAGE10;
		gPar.ProcessPosition.Stage[10]						:= POS_STAGE11;
		gPar.ProcessPosition.Stage[11]						:= POS_STAGE12;
		gPar.ProcessPosition.Stage[12]						:= POS_STAGE13;
		gPar.ProcessPosition.Stage[13]						:= POS_STAGE14;
		gPar.ProcessPosition.Stage[14]						:= POS_STAGE15;
		gPar.ProcessPosition.Stage[15]						:= POS_STAGE16;
		gPar.ProcessPosition.Stage[16]						:= POS_STAGE17;
		gPar.ProcessPosition.Stage[17]						:= POS_STAGE18;
		gPar.ProcessPosition.Stage[18]						:= POS_STAGE19;

		// Velocity Parameter Intialize
		gPar.MovementPar.Stage1.Velocity					:= 2.0;
		gPar.MovementPar.Stage1.Acceleration				:= 3.5;
		gPar.MovementPar.Stage1.Deceleration				:= 3.5;
		gPar.MovementPar.Stage1.MaxController				:= 1;

		gPar.MovementPar.Stage2.Velocity					:= 2.0;
		gPar.MovementPar.Stage2.Acceleration				:= 3.5;
		gPar.MovementPar.Stage2.Deceleration				:= 3.5;
		gPar.MovementPar.Stage2.MaxController				:= 1;

		gPar.MovementPar.Stage3.Velocity					:= 2.0;
		gPar.MovementPar.Stage3.Acceleration				:= 3.5;
		gPar.MovementPar.Stage3.Deceleration				:= 3.5;
		gPar.MovementPar.Stage3.MaxController				:= 1;

		gPar.MovementPar.Stage4.Velocity					:= 2.0;
		gPar.MovementPar.Stage4.Acceleration				:= 3.5;
		gPar.MovementPar.Stage4.Deceleration				:= 3.5;
		gPar.MovementPar.Stage4.MaxController				:= 1;

		gPar.MovementPar.Stage5.Velocity					:= 2.0;
		gPar.MovementPar.Stage5.Acceleration				:= 3.5;
		gPar.MovementPar.Stage5.Deceleration				:= 3.5;
		gPar.MovementPar.Stage5.MaxController				:= 1;

		gPar.MovementPar.Stage6.Velocity					:= 2.0;
		gPar.MovementPar.Stage6.Acceleration				:= 3.5;
		gPar.MovementPar.Stage6.Deceleration				:= 3.5;
		gPar.MovementPar.Stage6.MaxController				:= 1;

		gPar.MovementPar.Stage7.Velocity					:= 2.0;
		gPar.MovementPar.Stage7.Acceleration				:= 3.5;
		gPar.MovementPar.Stage7.Deceleration				:= 3.5;
		gPar.MovementPar.Stage7.MaxController				:= 1;

		gPar.MovementPar.Stage8.Velocity					:= 2.0;
		gPar.MovementPar.Stage8.Acceleration				:= 3.5;
		gPar.MovementPar.Stage8.Deceleration				:= 3.5;
		gPar.MovementPar.Stage8.MaxController				:= 1;

		gPar.MovementPar.Stage9.Velocity					:= 2.0;
		gPar.MovementPar.Stage9.Acceleration				:= 3.5;
		gPar.MovementPar.Stage9.Deceleration				:= 3.5;
		gPar.MovementPar.Stage9.MaxController				:= 1;
		// Maint
		gPar.MovementPar.Stage10.Velocity					:= 2.0;
		gPar.MovementPar.Stage10.Acceleration				:= 4.0;
		gPar.MovementPar.Stage10.Deceleration				:= 4.0;
		gPar.MovementPar.Stage10.MaxController				:= 3;

		gPar.MovementPar.Stage11.Velocity					:= 2.0;
		gPar.MovementPar.Stage11.Acceleration				:= 4.0;
		gPar.MovementPar.Stage11.Deceleration				:= 4.0;
		gPar.MovementPar.Stage11.MaxController				:= 1;

		gPar.MovementPar.Stage12.Velocity					:= 2.0;
		gPar.MovementPar.Stage12.Acceleration				:= 3.5;
		gPar.MovementPar.Stage12.Deceleration				:= 3.5;
		gPar.MovementPar.Stage12.MaxController				:= 1;

		gPar.MovementPar.Stage13.Velocity					:= 2.0;
		gPar.MovementPar.Stage13.Acceleration				:= 3.5;
		gPar.MovementPar.Stage13.Deceleration				:= 3.5;
		gPar.MovementPar.Stage13.MaxController				:= 1;

		gPar.MovementPar.Stage14.Velocity					:= 2.0;
		gPar.MovementPar.Stage14.Acceleration				:= 3.5;
		gPar.MovementPar.Stage14.Deceleration				:= 3.5;
		gPar.MovementPar.Stage14.MaxController				:= 2;

		gPar.MovementPar.Stage15.Velocity					:= 2.0;
		gPar.MovementPar.Stage15.Acceleration				:= 3.5;
		gPar.MovementPar.Stage15.Deceleration				:= 3.5;
		gPar.MovementPar.Stage15.MaxController				:= 1;

		gPar.MovementPar.Stage16.Velocity					:= 2.0;
		gPar.MovementPar.Stage16.Acceleration				:= 3.5;
		gPar.MovementPar.Stage16.Deceleration				:= 3.5;
		gPar.MovementPar.Stage16.MaxController				:= 1;

		gPar.MovementPar.Stage17.Velocity					:= 2.0;
		gPar.MovementPar.Stage17.Acceleration				:= 3.0;
		gPar.MovementPar.Stage17.Deceleration				:= 3.0;
		gPar.MovementPar.Stage17.MaxController				:= 1;

		gPar.MovementPar.Stage18.Velocity					:= 2.0;
		gPar.MovementPar.Stage18.Acceleration				:= 3.0;
		gPar.MovementPar.Stage18.Deceleration				:= 3.0;
		gPar.MovementPar.Stage18.MaxController				:= 2;

		gPar.MovementPar.Stage19.Velocity					:= 2.0;
		gPar.MovementPar.Stage19.Acceleration				:= 3.0;
		gPar.MovementPar.Stage19.Deceleration				:= 3.0;
		gPar.MovementPar.Stage19.MaxController				:= 1;

		gPar.MovementPar.Return.Velocity					:= 2.0;
		gPar.MovementPar.Return.RoutedVelocity				:= 2.0;
		gPar.MovementPar.Return.Acceleration				:= 3.5;
		gPar.MovementPar.Return.Deceleration				:= 3.5;

		gPar.TargetPPM 										:= 40;
		gPar.CountOfGroup 									:= 1;

		gParVision.Cam.MaxItemCnt	:= 1;
		gParVision.Cam.Timeout		:= 5000;
		gParVision.Cam.Gain			:= 1;
		gParVision.Cam.Focus		:= 20715;
		gParVision.Cam.Exposure		:= 14;
//		gParInitialized 									:= TRUE;
	END_IF
END_ACTION
```

### Program Logical/Source/Control/ifStage1 (IEC) - Can supply

#### Variables.var
```iecst
(**)
VAR
	currentProcess : E_PROCESS_STATUS;
	targetSlot : REFERENCE TO MyTrakSlotType;
	nextSlot : {REDUND_UNREPLICABLE} UDINT;
	shuttleID : REFERENCE TO STRING[19];
END_VAR
(**)
VAR
	step : DINT;
END_VAR
(**)
VAR
	interface : Interface_Process;
	userData : ShuttleUserData_typ;
END_VAR
(**)
VAR
	fbUserData : MC_BR_ShCopyUserData_AcpTrak;
END_VAR
(**)
VAR
	tmr : TON;
	fbShuttleOutCheck : MC_BR_TrgPointEnable_AcpTrak;
END_VAR
(**)
VAR
	NextReady : BOOL;
END_VAR
(**)
VAR
	bBlockSendOnce : BOOL;
	bBlockSendOnceAck : BOOL;
	bBlockReadOnce : BOOL;
	bBlockReadOnceAck : BOOL;
	bBlockSendShuttleID : BOOL;
	bBlockSendShuttleIDAck : BOOL;
END_VAR
```

#### Main.st
```iecst
PROGRAM _INIT
	currentProcess							:= E_PROCESS_Stage1;
	fbUserData.Axis							:= ADR(StStage[0].Shuttle);
	nextSlot 								:= ADR(StStage[1]);

	fbShuttleOutCheck.ProcessPoint			:= ADR(ptStage1);

	targetSlot ACCESS ADR(StStage[0]);
	shuttleID ACCESS ADR(interface.Trak.Data[0]);

	// Barrier for buffer
	BrBuffer.ProcessPoint := ADR(ptBuffer);

	BrBuffer.Command := mcACPTRAK_BARRIER_OPEN;
	BrBuffer.Execute := TRUE;

	BrBuffer();
END_PROGRAM

PROGRAM _CYCLIC
	IF gSim = TRUE THEN
		bBlockReadOnceAck := bBlockReadOnce;
		bBlockSendOnceAck := bBlockSendOnce;
		bBlockSendShuttleIDAck := bBlockSendShuttleID;

		IF interface.Trak.ShuttleArrived = TRUE THEN
			interface.Equipment.Ready 		:= FALSE;

			tmr.IN 							:= TRUE;
			tmr.PT 							:= T#1s;
		END_IF

		IF tmr.Q = TRUE THEN
			interface.Equipment.Data2[0]	:= interface.Equipment.Data2[0] + 1;
			interface.Equipment.Done 		:= TRUE;
		END_IF

		IF interface.Trak.ShuttleArrived = FALSE THEN
			tmr.IN							:= FALSE;
			interface.Equipment.Ready 		:= TRUE;
			interface.Equipment.Done 		:= FALSE;
		END_IF

		tmr();
	END_IF

	/////////////////////////////////////////////////////////////////
	// Barrier for Buffer
	IF gSts.AsmState = E_ASM_PROCESS THEN
		IF interface.Equipment.Ready THEN

			BrBuffer.Command := mcACPTRAK_BARRIER_OPEN;
			BrBuffer.Execute := TRUE;

		ELSIF interface.Equipment.Ready THEN

			BrBuffer.Command := mcACPTRAK_BARRIER_CLOSE;
			BrBuffer.Execute := TRUE;

		END_IF
	END_IF

	IF BrBuffer.Done THEN
		BrBuffer.Execute := FALSE;
	END_IF
	/////////////////////////////////////////////////////////////////

	IF targetSlot.Interface = E_SLOT_UNKNOWN THEN
		step 				:= 0;
	END_IF

	CASE step OF
		0:	(* Modbus Interface Initialize and Shuttle Check *)
			bBlockSendShuttleID					:= FALSE;
			bBlockSendOnce						:= FALSE;
			bBlockReadOnce						:= FALSE;

			//interface.Trak.ShuttleArrived		:= FALSE;

			IF targetSlot.Shuttle.controlif <> 0 AND bBlockSendOnceAck = FALSE AND bBlockReadOnceAck = FALSE AND bBlockSendShuttleIDAck = FALSE THEN
				step 							:= 10;
			END_IF

		10:	(* Read Shuttle Data from userData *)
			fbUserData.DataAddress 				:= ADR(userData);
			fbUserData.DataSize 				:= SIZEOF(userData);
			fbUserData.Mode						:= mcACPTRAK_USERDATA_GET;
			fbUserData.Execute 					:= TRUE;

			IF fbUserData.Done = TRUE THEN
				//End to Read Data fron user Data
				fbUserData.Execute 				:= FALSE;

				//Copy User Data to Modbus IO
				brsmemcpy(ADR(interface.Trak.Data[0]),ADR(userData.SerialNumber), 11);
				brsmemcpy(ADR(interface.Trak.Data2[0]),ADR(userData.Data[0]), SIZEOF(userData.Data));

				//Start to Write userdata to Modbus
				bBlockSendOnce					:= TRUE;
				bBlockSendShuttleID				:= TRUE;
				step 							:= 11;
			END_IF

		11: (* Check End of write to Modbus *)
			IF bBlockSendOnceAck AND bBlockSendShuttleIDAck THEN
				bBlockSendOnce					:= FALSE;
				bBlockSendShuttleID				:= FALSE;
				step							:= 20;
			END_IF

		20: (* Check Process Ready *)
			IF targetSlot.Interface = E_SLOT_PROCESS_READY THEN
				step 							:= 30;
			ELSIF targetSlot.Shuttle.controlif = 0 THEN
				step 							:= 0;
			END_IF

		30:	(* Check Assemble Status and Slot Status *)
			IF (gSts.AsmState = E_ASM_PROCESS OR gSts.AsmState = E_ASM_IDLE)
				AND targetSlot.Interface = E_SLOT_PROCESS_READY THEN
				interface.Trak.ShuttleArrived	:= TRUE;
				fbShuttleOutCheck.Enable		:= TRUE;
				step 							:= 100;
			END_IF

		100: (* Wait Proess End and Next Stage Ready *)
			IF interface.Equipment.Done = TRUE AND NextReady THEN
				//Start to Read Data from PLC
				bBlockReadOnce					:= TRUE;
				step 							:= 101;
			END_IF

		101:
			IF bBlockReadOnceAck = TRUE THEN
				// Save Current Process Status
				userData.ProcessStatus			:= currentProcess;

				// Read process data from PLC
				brsmemcpy(ADR(userData.Data[0]), ADR(interface.Equipment.Data2[0]), SIZEOF(interface.Equipment.Data2));

				// End to Read Data from PLC
				bBlockReadOnce					:= FALSE;
				step := 110;
			END_IF

		110: 	//Write User Data
			fbUserData.DataAddress 				:= ADR(userData);
			fbUserData.DataSize 				:= SIZE_OF_USERDATA;
			fbUserData.Mode						:= mcACPTRAK_USERDATA_SET;
			fbUserData.Execute 					:= TRUE;

			IF fbUserData.Done = TRUE THEN
				fbUserData.Execute 				:= FALSE;
				//	interface.Trak.ShuttleArrived 	:= FALSE;
				targetSlot.Interface 			:= E_SLOT_TAKEOUT_READY;
				targetSlot.NextStage			:= nextSlot;
				step 							:= 120;
			END_IF

		120: 	//Done Check
			IF interface.Equipment.Done = FALSE THEN
				step 						:= 0;
			END_IF
	END_CASE;

	IF fbShuttleOutCheck.EventCount > 0 THEN
		interface.Trak.ShuttleArrived	:= FALSE;
		fbShuttleOutCheck.Enable		:= FALSE;
	END_IF

	IF targetSlot.Shuttle.controlif = 0 AND shuttleID <> '' THEN
		brsmemset(ADR(interface.Trak.Data[0]),0,11);
	END_IF

	fbUserData();
	fbShuttleOutCheck();
	BrBuffer();
END_PROGRAM
```

### Program Logical/Source/Control/ifStage2 (IEC) - TC insert

#### Variables.var
```iecst
(**)
VAR
	currentProcess : E_PROCESS_STATUS;
	targetSlot : REFERENCE TO MyTrakSlotType;
	nextSlot : {REDUND_UNREPLICABLE} UDINT;
	shuttleID : REFERENCE TO STRING[19];
END_VAR
(**)
VAR
	step : DINT;
END_VAR
(**)
VAR
	interface : Interface_Process;
	userData : ShuttleUserData_typ;
END_VAR
(**)
VAR
	fbUserData : MC_BR_ShCopyUserData_AcpTrak;
END_VAR
(**)
VAR
	tmr : TON;
	fbShuttleOutCheck : MC_BR_TrgPointEnable_AcpTrak;
END_VAR
(**)
VAR
	NextReady : BOOL;
END_VAR
(**)
VAR
	Timer : TON;
	Timer2 : TON;
END_VAR
(**)
VAR
	bBlockSendOnce : BOOL;
	bBlockSendOnceAck : BOOL;
	bBlockReadOnce : BOOL;
	bBlockReadOnceAck : BOOL;
	bBlockSendShuttleID : BOOL;
	bBlockSendShuttleIDAck : BOOL;
END_VAR
```

#### Main.st
```iecst
PROGRAM _INIT
	currentProcess							:= E_PROCESS_Stage2;
	fbUserData.Axis							:= ADR(StStage[1].Shuttle);
	nextSlot 								:= ADR(StStage[2]);

	fbShuttleOutCheck.ProcessPoint			:= ADR(ptStage2);

	targetSlot ACCESS ADR(StStage[1]);
	shuttleID ACCESS ADR(interface.Trak.Data[0]);
END_PROGRAM

PROGRAM _CYCLIC
	IF gSim = TRUE THEN
		bBlockReadOnceAck := bBlockReadOnce;
		bBlockSendOnceAck := bBlockSendOnce;
		bBlockSendShuttleIDAck := bBlockSendShuttleID;

		interface.Equipment.Data2[0]	:= interface.Trak.Data2[0];

		IF interface.Trak.ShuttleArrived = TRUE THEN
			interface.Equipment.Ready 		:= FALSE;

			tmr.IN 							:= TRUE;
			tmr.PT 							:= T#1s;
		END_IF

		IF tmr.Q = TRUE THEN
			interface.Equipment.Done 		:= TRUE;
		END_IF

		IF interface.Trak.ShuttleArrived = FALSE THEN
			tmr.IN							:= FALSE;
			interface.Equipment.Ready 		:= TRUE;
			interface.Equipment.Done 		:= FALSE;
		END_IF

		tmr();
	END_IF

	IF targetSlot.Interface = E_SLOT_UNKNOWN THEN
		step 				:= 0;
	END_IF

	CASE step OF
		0:	(* Modbus Interface Initialize and Shuttle Check *)
			bBlockSendShuttleID					:= FALSE;
			bBlockSendOnce						:= FALSE;
			bBlockReadOnce						:= FALSE;

			//interface.Trak.ShuttleArrived		:= FALSE;

			IF targetSlot.Shuttle.controlif <> 0 AND bBlockSendOnceAck = FALSE AND bBlockReadOnceAck = FALSE AND bBlockSendShuttleIDAck = FALSE THEN
				step 							:= 10;
			END_IF

		10:	(* Read Shuttle Data from userData *)
			fbUserData.DataAddress 				:= ADR(userData);
			fbUserData.DataSize 				:= SIZEOF(userData);
			fbUserData.Mode						:= mcACPTRAK_USERDATA_GET;
			fbUserData.Execute 					:= TRUE;

			IF fbUserData.Done = TRUE THEN
				//End to Read Data fron user Data
				fbUserData.Execute 				:= FALSE;

				//Copy User Data to Modbus IO
				brsmemcpy(ADR(interface.Trak.Data[0]),ADR(userData.SerialNumber), 11);
				brsmemcpy(ADR(interface.Trak.Data2[0]),ADR(userData.Data[0]), SIZEOF(userData.Data));

				//Start to Write userdata to Modbus
				bBlockSendOnce					:= TRUE;
				bBlockSendShuttleID				:= TRUE;
				step 							:= 11;
			END_IF

		11: (* Check End of write to Modbus *)
			IF bBlockSendOnceAck AND bBlockSendShuttleIDAck THEN
				bBlockSendOnce					:= FALSE;
				bBlockSendShuttleID				:= FALSE;
				step							:= 20;
			END_IF

		20: (* Check Process Ready *)
			IF targetSlot.Interface = E_SLOT_PROCESS_READY THEN
				step 							:= 30;
			ELSIF targetSlot.Shuttle.controlif = 0 THEN
				step 							:= 0;
			END_IF

		30:	(* Check Assemble Status and Slot Status *)
			IF (gSts.AsmState = E_ASM_PROCESS OR gSts.AsmState = E_ASM_IDLE)
				AND targetSlot.Interface = E_SLOT_PROCESS_READY THEN
				interface.Trak.ShuttleArrived	:= TRUE;
				fbShuttleOutCheck.Enable		:= TRUE;
				step 							:= 100;
			END_IF

		100: (* Wait Proess End and Next Stage Ready *)
			IF interface.Equipment.Done = TRUE AND NextReady THEN
				//Start to Read Data from PLC
				bBlockReadOnce					:= TRUE;
				step 							:= 101;
			END_IF

		101:
			IF bBlockReadOnceAck = TRUE THEN
				// Save Current Process Status
				userData.ProcessStatus			:= currentProcess;

				// Read process data from PLC
				brsmemcpy(ADR(userData.Data[0]), ADR(interface.Equipment.Data2[0]), SIZEOF(interface.Equipment.Data2));

				// End to Read Data from PLC
				bBlockReadOnce					:= FALSE;
				step := 110;
			END_IF

		110: 	//Write User Data
			fbUserData.DataAddress 				:= ADR(userData);
			fbUserData.DataSize 				:= SIZE_OF_USERDATA;
			fbUserData.Mode						:= mcACPTRAK_USERDATA_SET;
			fbUserData.Execute 					:= TRUE;

			IF fbUserData.Done = TRUE THEN
				fbUserData.Execute 				:= FALSE;
				//	interface.Trak.ShuttleArrived 	:= FALSE;
				targetSlot.Interface 			:= E_SLOT_TAKEOUT_READY;
				targetSlot.NextStage			:= nextSlot;
				step 							:= 120;
			END_IF

		120: 	//Done Check
			IF interface.Equipment.Done = FALSE THEN
				step 						:= 0;
			END_IF
	END_CASE;

	IF fbShuttleOutCheck.EventCount > 0 THEN
		interface.Trak.ShuttleArrived	:= FALSE;
		fbShuttleOutCheck.Enable		:= FALSE;
	END_IF

	IF targetSlot.Shuttle.controlif = 0 AND shuttleID <> '' THEN
		brsmemset(ADR(interface.Trak.Data[0]),0,11);
	END_IF

	fbUserData();
	fbShuttleOutCheck();
END_PROGRAM
```

### Program Logical/Source/Control/ifStage3 (IEC) - TC push

#### Main.st
```iecst
PROGRAM _INIT
	currentProcess							:= E_PROCESS_Stage3;
	fbUserData.Axis							:= ADR(StStage[2].Shuttle);
	nextSlot 								:= ADR(StStage[3]);

	fbShuttleOutCheck.ProcessPoint			:= ADR(ptStage3);

	targetSlot ACCESS ADR(StStage[2]);
	shuttleID ACCESS ADR(interface.Trak.Data[0]);
END_PROGRAM

PROGRAM _CYCLIC
	IF gSim = TRUE THEN
		bBlockReadOnceAck := bBlockReadOnce;
		bBlockSendOnceAck := bBlockSendOnce;
		bBlockSendShuttleIDAck := bBlockSendShuttleID;

		IF interface.Trak.ShuttleArrived = TRUE THEN
			interface.Equipment.Ready 		:= FALSE;

			tmr.IN 							:= TRUE;
			tmr.PT 							:= T#1s;
		END_IF

		IF tmr.Q = TRUE THEN
			interface.Equipment.Done 		:= TRUE;
		END_IF

		IF interface.Trak.ShuttleArrived = FALSE THEN
			tmr.IN							:= FALSE;
			interface.Equipment.Ready 		:= TRUE;
			interface.Equipment.Done 		:= FALSE;
		END_IF

		tmr();
	END_IF

	IF targetSlot.Interface = E_SLOT_UNKNOWN THEN
		step 				:= 0;
	END_IF

	CASE step OF
		0:	(* Modbus Interface Initialize and Shuttle Check *)
			bBlockSendShuttleID					:= FALSE;
			bBlockSendOnce						:= FALSE;
			bBlockReadOnce						:= FALSE;

			//interface.Trak.ShuttleArrived		:= FALSE;

			IF targetSlot.Shuttle.controlif <> 0 AND bBlockSendOnceAck = FALSE AND bBlockReadOnceAck = FALSE AND bBlockSendShuttleIDAck = FALSE THEN
				step 							:= 10;
			END_IF

		10:	(* Read Shuttle Data from userData *)
			fbUserData.DataAddress 				:= ADR(userData);
			fbUserData.DataSize 				:= SIZEOF(userData);
			fbUserData.Mode						:= mcACPTRAK_USERDATA_GET;
			fbUserData.Execute 					:= TRUE;

			IF fbUserData.Done = TRUE THEN
				//End to Read Data fron user Data
				fbUserData.Execute 				:= FALSE;

				//Copy User Data to Modbus IO
				brsmemcpy(ADR(interface.Trak.Data[0]),ADR(userData.SerialNumber), 11);
				brsmemcpy(ADR(interface.Trak.Data2[0]),ADR(userData.Data[0]), SIZEOF(userData.Data));

				//Start to Write userdata to Modbus
				bBlockSendOnce					:= TRUE;
				bBlockSendShuttleID				:= TRUE;
				step 							:= 11;
			END_IF

		11: (* Check End of write to Modbus *)
			IF bBlockSendOnceAck AND bBlockSendShuttleIDAck THEN
				bBlockSendOnce					:= FALSE;
				bBlockSendShuttleID				:= FALSE;
				step							:= 20;
			END_IF

		20: (* Check Process Ready *)
			IF targetSlot.Interface = E_SLOT_PROCESS_READY THEN
				step 							:= 30;
			ELSIF targetSlot.Shuttle.controlif = 0 THEN
				step 							:= 0;
			END_IF

		30:	(* Check Assemble Status and Slot Status *)
			IF (gSts.AsmState = E_ASM_PROCESS OR gSts.AsmState = E_ASM_IDLE)
				AND targetSlot.Interface = E_SLOT_PROCESS_READY THEN
				interface.Trak.ShuttleArrived	:= TRUE;
				fbShuttleOutCheck.Enable		:= TRUE;
				step 							:= 100;
			END_IF

		100: (* Wait Proess End and Next Stage Ready *)
			IF interface.Equipment.Done = TRUE AND NextReady THEN
				//Start to Read Data from PLC
				bBlockReadOnce					:= TRUE;
				step 							:= 101;
			END_IF

		101:
			IF bBlockReadOnceAck = TRUE THEN
				// Save Current Process Status
				userData.ProcessStatus			:= currentProcess;

				// Read process data from PLC
				brsmemcpy(ADR(userData.Data[0]), ADR(interface.Equipment.Data2[0]), SIZEOF(interface.Equipment.Data2));

				// End to Read Data from PLC
				bBlockReadOnce					:= FALSE;
				step := 110;
			END_IF

		110: 	//Write User Data
			fbUserData.DataAddress 				:= ADR(userData);
			fbUserData.DataSize 				:= SIZE_OF_USERDATA;
			fbUserData.Mode						:= mcACPTRAK_USERDATA_SET;
			fbUserData.Execute 					:= TRUE;

			IF fbUserData.Done = TRUE THEN
				fbUserData.Execute 				:= FALSE;
				//	interface.Trak.ShuttleArrived 	:= FALSE;
				targetSlot.Interface 			:= E_SLOT_TAKEOUT_READY;
				targetSlot.NextStage			:= nextSlot;
				step 							:= 120;
			END_IF

		120: 	//Done Check
			IF interface.Equipment.Done = FALSE THEN
				step 						:= 0;
			END_IF
	END_CASE;

	IF fbShuttleOutCheck.EventCount > 0 THEN
		interface.Trak.ShuttleArrived	:= FALSE;
		fbShuttleOutCheck.Enable		:= FALSE;
	END_IF

	IF targetSlot.Shuttle.controlif = 0 AND shuttleID <> '' THEN
		brsmemset(ADR(interface.Trak.Data[0]),0,11);
	END_IF

	fbUserData();
	fbShuttleOutCheck();
	Timer();
	Timer2();

END_PROGRAM
```

### Program Logical/Source/Control/ifStage4 (IEC) - TC vision

#### Main.st
```iecst
PROGRAM _INIT
	currentProcess							:= E_PROCESS_Stage4;
	fbUserData.Axis							:= ADR(StStage[3].Shuttle);
	nextSlot 								:= ADR(StStage[4]);

	fbShuttleOutCheck.ProcessPoint			:= ADR(ptStage4);

	targetSlot ACCESS ADR(StStage[3]);
	shuttleID ACCESS ADR(interface.Trak.Data[0]);
END_PROGRAM

PROGRAM _CYCLIC
	IF gSim = TRUE THEN
		bBlockReadOnceAck := bBlockReadOnce;
		bBlockSendOnceAck := bBlockSendOnce;
		bBlockSendShuttleIDAck := bBlockSendShuttleID;

		IF interface.Trak.ShuttleArrived = TRUE THEN
			interface.Equipment.Ready 		:= FALSE;

			tmr.IN 							:= TRUE;
			tmr.PT 							:= T#1s;
		END_IF

		IF tmr.Q = TRUE THEN
			interface.Equipment.Done 		:= TRUE;
		END_IF

		IF interface.Trak.ShuttleArrived = FALSE THEN
			tmr.IN							:= FALSE;
			interface.Equipment.Ready 		:= TRUE;
			interface.Equipment.Done 		:= FALSE;
		END_IF

		tmr();
	END_IF

	IF targetSlot.Interface = E_SLOT_UNKNOWN THEN
		step 				:= 0;
	END_IF

	CASE step OF
		0:	(* Modbus Interface Initialize and Shuttle Check *)
			bBlockSendShuttleID					:= FALSE;
			bBlockSendOnce						:= FALSE;
			bBlockReadOnce						:= FALSE;

			//interface.Trak.ShuttleArrived		:= FALSE;

			IF targetSlot.Shuttle.controlif <> 0 AND bBlockSendOnceAck = FALSE AND bBlockReadOnceAck = FALSE AND bBlockSendShuttleIDAck = FALSE THEN
				step 							:= 10;
			END_IF

		10:	(* Read Shuttle Data from userData *)
			fbUserData.DataAddress 				:= ADR(userData);
			fbUserData.DataSize 				:= SIZEOF(userData);
			fbUserData.Mode						:= mcACPTRAK_USERDATA_GET;
			fbUserData.Execute 					:= TRUE;

			IF fbUserData.Done = TRUE THEN
				//End to Read Data fron user Data
				fbUserData.Execute 				:= FALSE;

				//Copy User Data to Modbus IO
				brsmemcpy(ADR(interface.Trak.Data[0]),ADR(userData.SerialNumber), 11);
				brsmemcpy(ADR(interface.Trak.Data2[0]),ADR(userData.Data[0]), SIZEOF(userData.Data));

				//Start to Write userdata to Modbus
				bBlockSendOnce					:= TRUE;
				bBlockSendShuttleID				:= TRUE;
				step 							:= 11;
			END_IF

		11: (* Check End of write to Modbus *)
			IF bBlockSendOnceAck AND bBlockSendShuttleIDAck THEN
				bBlockSendOnce					:= FALSE;
				bBlockSendShuttleID				:= FALSE;
				step							:= 20;
			END_IF

		20: (* Check Process Ready *)
			IF targetSlot.Interface = E_SLOT_PROCESS_READY THEN
				step 							:= 30;
			ELSIF targetSlot.Shuttle.controlif = 0 THEN
				step 							:= 0;
			END_IF

		30:	(* Check Assemble Status and Slot Status *)
			IF (gSts.AsmState = E_ASM_PROCESS OR gSts.AsmState = E_ASM_IDLE)
				AND targetSlot.Interface = E_SLOT_PROCESS_READY THEN
				interface.Trak.ShuttleArrived	:= TRUE;
				fbShuttleOutCheck.Enable		:= TRUE;
				step 							:= 100;
			END_IF

		100: (* Wait Proess End and Next Stage Ready *)
			IF interface.Equipment.Done = TRUE AND NextReady THEN
				//Start to Read Data from PLC
				bBlockReadOnce					:= TRUE;
				step 							:= 101;
			END_IF

		101:
			IF bBlockReadOnceAck = TRUE THEN
				// Save Current Process Status
				userData.ProcessStatus			:= currentProcess;

				// Read process data from PLC
				brsmemcpy(ADR(userData.Data[0]), ADR(interface.Equipment.Data2[0]), SIZEOF(interface.Equipment.Data2));

				// End to Read Data from PLC
				bBlockReadOnce					:= FALSE;
				step := 110;
			END_IF

		110: 	//Write User Data
			fbUserData.DataAddress 				:= ADR(userData);
			fbUserData.DataSize 				:= SIZE_OF_USERDATA;
			fbUserData.Mode						:= mcACPTRAK_USERDATA_SET;
			fbUserData.Execute 					:= TRUE;

			IF fbUserData.Done = TRUE THEN
				fbUserData.Execute 				:= FALSE;
				//	interface.Trak.ShuttleArrived 	:= FALSE;
				targetSlot.Interface 			:= E_SLOT_TAKEOUT_READY;
				targetSlot.NextStage			:= nextSlot;
				step 							:= 120;
			END_IF

		120: 	//Done Check
			IF interface.Equipment.Done = FALSE THEN
				step 						:= 0;
			END_IF
	END_CASE;

	IF fbShuttleOutCheck.EventCount > 0 THEN
		interface.Trak.ShuttleArrived	:= FALSE;
		fbShuttleOutCheck.Enable		:= FALSE;
	END_IF

	IF targetSlot.Shuttle.controlif = 0 AND shuttleID <> '' THEN
		brsmemset(ADR(interface.Trak.Data[0]),0,11);
	END_IF

	fbUserData();
	fbShuttleOutCheck();
	Timer();
	Timer2();

END_PROGRAM
```

### Program Logical/Source/Control/ifStage5 (IEC) - TC NG re-insert

#### Main.st
```iecst
PROGRAM _INIT
	currentProcess							:= E_PROCESS_Stage5;
	fbUserData.Axis							:= ADR(StStage[4].Shuttle);
	nextSlot 								:= ADR(StStage[5]);

	fbShuttleOutCheck.ProcessPoint			:= ADR(ptStage5);

	targetSlot ACCESS ADR(StStage[4]);
	shuttleID ACCESS ADR(interface.Trak.Data[0]);
END_PROGRAM

PROGRAM _CYCLIC
	IF gSim = TRUE THEN
		bBlockReadOnceAck := bBlockReadOnce;
		bBlockSendOnceAck := bBlockSendOnce;
		bBlockSendShuttleIDAck := bBlockSendShuttleID;

		IF interface.Trak.ShuttleArrived = TRUE THEN
			interface.Equipment.Ready 		:= FALSE;

			tmr.IN 							:= TRUE;
			tmr.PT 							:= T#1s;
		END_IF

		IF tmr.Q = TRUE THEN
			interface.Equipment.Done 		:= TRUE;
		END_IF

		IF interface.Trak.ShuttleArrived = FALSE THEN
			tmr.IN							:= FALSE;
			interface.Equipment.Ready 		:= TRUE;
			interface.Equipment.Done 		:= FALSE;
		END_IF

		tmr();
	END_IF

	IF targetSlot.Interface = E_SLOT_UNKNOWN THEN
		step 				:= 0;
	END_IF

	CASE step OF
		0:	(* Modbus Interface Initialize and Shuttle Check *)
			bBlockSendShuttleID					:= FALSE;
			bBlockSendOnce						:= FALSE;
			bBlockReadOnce						:= FALSE;

			//interface.Trak.ShuttleArrived		:= FALSE;

			IF targetSlot.Shuttle.controlif <> 0 AND bBlockSendOnceAck = FALSE AND bBlockReadOnceAck = FALSE AND bBlockSendShuttleIDAck = FALSE THEN
				step 							:= 10;
			END_IF

		10:	(* Read Shuttle Data from userData *)
			fbUserData.DataAddress 				:= ADR(userData);
			fbUserData.DataSize 				:= SIZEOF(userData);
			fbUserData.Mode						:= mcACPTRAK_USERDATA_GET;
			fbUserData.Execute 					:= TRUE;

			IF fbUserData.Done = TRUE THEN
				//End to Read Data fron user Data
				fbUserData.Execute 				:= FALSE;

				//Copy User Data to Modbus IO
				brsmemcpy(ADR(interface.Trak.Data[0]),ADR(userData.SerialNumber), 11);
				brsmemcpy(ADR(interface.Trak.Data2[0]),ADR(userData.Data[0]), SIZEOF(userData.Data));

				//Start to Write userdata to Modbus
				bBlockSendOnce					:= TRUE;
				bBlockSendShuttleID				:= TRUE;
				step 							:= 11;
			END_IF

		11: (* Check End of write to Modbus *)
			IF bBlockSendOnceAck AND bBlockSendShuttleIDAck THEN
				bBlockSendOnce					:= FALSE;
				bBlockSendShuttleID				:= FALSE;
				step							:= 20;
			END_IF

		20: (* Check Process Ready *)
			IF targetSlot.Interface = E_SLOT_PROCESS_READY THEN
				step 							:= 30;
			ELSIF targetSlot.Shuttle.controlif = 0 THEN
				step 							:= 0;
			END_IF

		30:	(* Check Assemble Status and Slot Status *)
			IF (gSts.AsmState = E_ASM_PROCESS OR gSts.AsmState = E_ASM_IDLE)
				AND targetSlot.Interface = E_SLOT_PROCESS_READY THEN
				interface.Trak.ShuttleArrived	:= TRUE;
				fbShuttleOutCheck.Enable		:= TRUE;
				step 							:= 100;
			END_IF

		100: (* Wait Proess End and Next Stage Ready *)
			IF interface.Equipment.Done = TRUE AND NextReady THEN
				//Start to Read Data from PLC
				bBlockReadOnce					:= TRUE;
				step 							:= 101;
			END_IF

		101:
			IF bBlockReadOnceAck = TRUE THEN
				// Save Current Process Status
				userData.ProcessStatus			:= currentProcess;

				// Read process data from PLC
				brsmemcpy(ADR(userData.Data[0]), ADR(interface.Equipment.Data2[0]), SIZEOF(interface.Equipment.Data2));

				// End to Read Data from PLC
				bBlockReadOnce					:= FALSE;
				step := 110;
			END_IF

		110: 	//Write User Data
			fbUserData.DataAddress 				:= ADR(userData);
			fbUserData.DataSize 				:= SIZE_OF_USERDATA;
			fbUserData.Mode						:= mcACPTRAK_USERDATA_SET;
			fbUserData.Execute 					:= TRUE;

			IF fbUserData.Done = TRUE THEN
				fbUserData.Execute 				:= FALSE;
				//	interface.Trak.ShuttleArrived 	:= FALSE;
				targetSlot.Interface 			:= E_SLOT_TAKEOUT_READY;
				targetSlot.NextStage			:= nextSlot;
				step 							:= 120;
			END_IF

		120: 	//Done Check
			IF interface.Equipment.Done = FALSE THEN
				step 						:= 0;
			END_IF
	END_CASE;

	IF fbShuttleOutCheck.EventCount > 0 THEN
		interface.Trak.ShuttleArrived	:= FALSE;
		fbShuttleOutCheck.Enable		:= FALSE;
	END_IF

	IF targetSlot.Shuttle.controlif = 0 AND shuttleID <> '' THEN
		brsmemset(ADR(interface.Trak.Data[0]),0,11);
	END_IF

	fbUserData();
	fbShuttleOutCheck();
	Timer();
	Timer2();

END_PROGRAM
```

### Program Logical/Source/Control/ifStage6 (IEC) - BCR vision

#### Main.st
```iecst
PROGRAM _INIT
	currentProcess							:= E_PROCESS_Stage6;
	fbUserData.Axis							:= ADR(StStage[5].Shuttle);
	nextSlot 								:= ADR(StStage[6]);

	fbShuttleOutCheck.ProcessPoint			:= ADR(ptStage6);

	targetSlot ACCESS ADR(StStage[5]);
	shuttleID ACCESS ADR(interface.Trak.Data[0]);
END_PROGRAM

PROGRAM _CYCLIC
	IF gSim = TRUE THEN
		bBlockReadOnceAck := bBlockReadOnce;
		bBlockSendOnceAck := bBlockSendOnce;
		bBlockSendShuttleIDAck := bBlockSendShuttleID;

		IF interface.Trak.ShuttleArrived = TRUE THEN
			interface.Equipment.Ready 		:= FALSE;

			tmr.IN 							:= TRUE;
			tmr.PT 							:= T#1s;
		END_IF

		IF tmr.Q = TRUE THEN
			interface.Equipment.Done 		:= TRUE;
		END_IF

		IF interface.Trak.ShuttleArrived = FALSE THEN
			tmr.IN							:= FALSE;
			interface.Equipment.Ready 		:= TRUE;
			interface.Equipment.Done 		:= FALSE;
		END_IF

		tmr();
	END_IF

	IF targetSlot.Interface = E_SLOT_UNKNOWN THEN
		step 				:= 0;
	END_IF

	CASE step OF
		0:	(* Modbus Interface Initialize and Shuttle Check *)
			bBlockSendShuttleID					:= FALSE;
			bBlockSendOnce						:= FALSE;
			bBlockReadOnce						:= FALSE;

			//interface.Trak.ShuttleArrived		:= FALSE;

			IF targetSlot.Shuttle.controlif <> 0 AND bBlockSendOnceAck = FALSE AND bBlockReadOnceAck = FALSE AND bBlockSendShuttleIDAck = FALSE THEN
				step 							:= 10;
			END_IF

		10:	(* Read Shuttle Data from userData *)
			fbUserData.DataAddress 				:= ADR(userData);
			fbUserData.DataSize 				:= SIZEOF(userData);
			fbUserData.Mode						:= mcACPTRAK_USERDATA_GET;
			fbUserData.Execute 					:= TRUE;

			IF fbUserData.Done = TRUE THEN
				//End to Read Data fron user Data
				fbUserData.Execute 				:= FALSE;

				//Copy User Data to Modbus IO
				brsmemcpy(ADR(interface.Trak.Data[0]),ADR(userData.SerialNumber), 11);
				brsmemcpy(ADR(interface.Trak.Data2[0]),ADR(userData.Data[0]), SIZEOF(userData.Data));

				//Start to Write userdata to Modbus
				bBlockSendOnce					:= TRUE;
				bBlockSendShuttleID				:= TRUE;
				step 							:= 11;
			END_IF

		11: (* Check End of write to Modbus *)
			IF bBlockSendOnceAck AND bBlockSendShuttleIDAck THEN
				bBlockSendOnce					:= FALSE;
				bBlockSendShuttleID				:= FALSE;
				step							:= 20;
			END_IF

		20: (* Check Process Ready *)
			IF targetSlot.Interface = E_SLOT_PROCESS_READY THEN
				step 							:= 30;
			ELSIF targetSlot.Shuttle.controlif = 0 THEN
				step 							:= 0;
			END_IF

		30:	(* Check Assemble Status and Slot Status *)
			IF (gSts.AsmState = E_ASM_PROCESS OR gSts.AsmState = E_ASM_IDLE)
				AND targetSlot.Interface = E_SLOT_PROCESS_READY THEN
				interface.Trak.ShuttleArrived	:= TRUE;
				fbShuttleOutCheck.Enable		:= TRUE;
				step 							:= 100;
			END_IF

		100: (* Wait Proess End and Next Stage Ready *)
			IF interface.Equipment.Done = TRUE AND NextReady THEN
				//Start to Read Data from PLC
				bBlockReadOnce					:= TRUE;
				step 							:= 101;
			END_IF

		101:
			IF bBlockReadOnceAck = TRUE THEN
				// Save Current Process Status
				userData.ProcessStatus			:= currentProcess;

				// Read process data from PLC
				brsmemcpy(ADR(userData.Data[0]), ADR(interface.Equipment.Data2[0]), SIZEOF(interface.Equipment.Data2));

				// End to Read Data from PLC
				bBlockReadOnce					:= FALSE;
				step := 110;
			END_IF

		110: 	//Write User Data
			fbUserData.DataAddress 				:= ADR(userData);
			fbUserData.DataSize 				:= SIZE_OF_USERDATA;
			fbUserData.Mode						:= mcACPTRAK_USERDATA_SET;
			fbUserData.Execute 					:= TRUE;

			IF fbUserData.Done = TRUE THEN
				fbUserData.Execute 				:= FALSE;
				//	interface.Trak.ShuttleArrived 	:= FALSE;
				targetSlot.Interface 			:= E_SLOT_TAKEOUT_READY;
				targetSlot.NextStage			:= nextSlot;
				step 							:= 120;
			END_IF

		120: 	//Done Check
			IF interface.Equipment.Done = FALSE THEN
				step 						:= 0;
			END_IF
	END_CASE;

	IF fbShuttleOutCheck.EventCount > 0 THEN
		interface.Trak.ShuttleArrived	:= FALSE;
		fbShuttleOutCheck.Enable		:= FALSE;
	END_IF

	IF targetSlot.Shuttle.controlif = 0 AND shuttleID <> '' THEN
		brsmemset(ADR(interface.Trak.Data[0]),0,11);
	END_IF

	fbUserData();
	fbShuttleOutCheck();
	Timer();
	Timer2();

END_PROGRAM
```

### Program Logical/Source/Control/ifStage7 (IEC) - CCR 1

#### Main.st
```iecst
PROGRAM _INIT
	currentProcess							:= E_PROCESS_Stage7;
	fbUserData.Axis							:= ADR(StStage[6].Shuttle);
	nextSlot 								:= ADR(StStage[7]);

	fbShuttleOutCheck.ProcessPoint			:= ADR(ptStage7);

	targetSlot ACCESS ADR(StStage[6]);
	shuttleID ACCESS ADR(interface.Trak.Data[0]);
END_PROGRAM

PROGRAM _CYCLIC
	IF gSim = TRUE THEN
		bBlockReadOnceAck := bBlockReadOnce;
		bBlockSendOnceAck := bBlockSendOnce;
		bBlockSendShuttleIDAck := bBlockSendShuttleID;

		IF interface.Trak.ShuttleArrived = TRUE THEN
			interface.Equipment.Ready 		:= FALSE;

			tmr.IN 							:= TRUE;
			tmr.PT 							:= T#1s;
		END_IF

		IF tmr.Q = TRUE THEN
			interface.Equipment.Done 		:= TRUE;
		END_IF

		IF interface.Trak.ShuttleArrived = FALSE THEN
			tmr.IN							:= FALSE;
			interface.Equipment.Ready 		:= TRUE;
			interface.Equipment.Done 		:= FALSE;
		END_IF

		tmr();
	END_IF

	IF targetSlot.Interface = E_SLOT_UNKNOWN THEN
		step 				:= 0;
	END_IF

	CASE step OF
		0:	(* Modbus Interface Initialize and Shuttle Check *)
			bBlockSendShuttleID					:= FALSE;
			bBlockSendOnce						:= FALSE;
			bBlockReadOnce						:= FALSE;

			//interface.Trak.ShuttleArrived		:= FALSE;

			IF targetSlot.Shuttle.controlif <> 0 AND bBlockSendOnceAck = FALSE AND bBlockReadOnceAck = FALSE AND bBlockSendShuttleIDAck = FALSE THEN
				step 							:= 10;
			END_IF

		10:	(* Read Shuttle Data from userData *)
			fbUserData.DataAddress 				:= ADR(userData);
			fbUserData.DataSize 				:= SIZEOF(userData);
			fbUserData.Mode						:= mcACPTRAK_USERDATA_GET;
			fbUserData.Execute 					:= TRUE;

			IF fbUserData.Done = TRUE THEN
				//End to Read Data fron user Data
				fbUserData.Execute 				:= FALSE;

				//Copy User Data to Modbus IO
				brsmemcpy(ADR(interface.Trak.Data[0]),ADR(userData.SerialNumber), 11);
				brsmemcpy(ADR(interface.Trak.Data2[0]),ADR(userData.Data[0]), SIZEOF(userData.Data));

				//Start to Write userdata to Modbus
				bBlockSendOnce					:= TRUE;
				bBlockSendShuttleID				:= TRUE;
				step 							:= 11;
			END_IF

		11: (* Check End of write to Modbus *)
			IF bBlockSendOnceAck AND bBlockSendShuttleIDAck THEN
				bBlockSendOnce					:= FALSE;
				bBlockSendShuttleID				:= FALSE;
				step							:= 20;
			END_IF

		20: (* Check Process Ready *)
			IF targetSlot.Interface = E_SLOT_PROCESS_READY THEN
				step 							:= 30;
			ELSIF targetSlot.Shuttle.controlif = 0 THEN
				step 							:= 0;
			END_IF

		30:	(* Check Assemble Status and Slot Status *)
			IF (gSts.AsmState = E_ASM_PROCESS OR gSts.AsmState = E_ASM_IDLE)
				AND targetSlot.Interface = E_SLOT_PROCESS_READY THEN
				interface.Trak.ShuttleArrived	:= TRUE;
				fbShuttleOutCheck.Enable		:= TRUE;
				step 							:= 100;
			END_IF

		100: (* Wait Proess End and Next Stage Ready *)
			IF interface.Equipment.Done = TRUE AND NextReady THEN
				//Start to Read Data from PLC
				bBlockReadOnce					:= TRUE;
				step 							:= 101;
			END_IF

		101:
			IF bBlockReadOnceAck = TRUE THEN
				// Save Current Process Status
				userData.ProcessStatus			:= currentProcess;

				// Read process data from PLC
				brsmemcpy(ADR(userData.Data[0]), ADR(interface.Equipment.Data2[0]), SIZEOF(interface.Equipment.Data2));

				// End to Read Data from PLC
				bBlockReadOnce					:= FALSE;
				step := 110;
			END_IF

		110: 	//Write User Data
			fbUserData.DataAddress 				:= ADR(userData);
			fbUserData.DataSize 				:= SIZE_OF_USERDATA;
			fbUserData.Mode						:= mcACPTRAK_USERDATA_SET;
			fbUserData.Execute 					:= TRUE;

			IF fbUserData.Done = TRUE THEN
				fbUserData.Execute 				:= FALSE;
				//	interface.Trak.ShuttleArrived 	:= FALSE;
				targetSlot.Interface 			:= E_SLOT_TAKEOUT_READY;
				targetSlot.NextStage			:= nextSlot;
				step 							:= 120;
			END_IF

		120: 	//Done Check
			IF interface.Equipment.Done = FALSE THEN
				step 						:= 0;
			END_IF
	END_CASE;

	IF fbShuttleOutCheck.EventCount > 0 THEN
		interface.Trak.ShuttleArrived	:= FALSE;
		fbShuttleOutCheck.Enable		:= FALSE;
	END_IF

	IF targetSlot.Shuttle.controlif = 0 AND shuttleID <> '' THEN
		brsmemset(ADR(interface.Trak.Data[0]),0,11);
	END_IF

	fbUserData();
	fbShuttleOutCheck();
	Timer();
	Timer2();

END_PROGRAM
```

### Program Logical/Source/Control/ifStage8 (IEC) - CCR 1 vision

#### Variables.var
```iecst
(**)
VAR
	currentProcess : E_PROCESS_STATUS;
	targetSlot : REFERENCE TO MyTrakSlotType;
	nextSlot : {REDUND_UNREPLICABLE} UDINT;
	shuttleID : REFERENCE TO STRING[19];
END_VAR
(**)
VAR
	step : DINT;
END_VAR
(**)
VAR
	interface : Interface_Process;
	userData : ShuttleUserData_typ;
END_VAR
(**)
VAR
	fbUserData : MC_BR_ShCopyUserData_AcpTrak;
END_VAR
(**)
VAR
	tmr : TON;
	fbShuttleOutCheck : MC_BR_TrgPointEnable_AcpTrak;
END_VAR
(**)
VAR
	NextReady : BOOL;
	Timer : TON;
	Timer2 : TON;
END_VAR
(**)
VAR
	bBlockSendOnce : BOOL;
	bBlockSendOnceAck : BOOL;
	bBlockReadOnce : BOOL;
	bBlockReadOnceAck : BOOL;
	bBlockSendShuttleID : BOOL;
	bBlockSendShuttleIDAck : BOOL;
END_VAR
(**)
VAR
	ParStringTmp : STRING[80];
	ParString : WSTRING[80];
	auditTag : WSTRING[80];
END_VAR
```

#### Main.st
```iecst
PROGRAM _INIT
	currentProcess							:= E_PROCESS_Stage8;
	fbUserData.Axis							:= ADR(StStage[7].Shuttle);
	nextSlot 								:= ADR(StStage[8]);

	fbShuttleOutCheck.ProcessPoint			:= ADR(ptStage8);

	targetSlot ACCESS ADR(StStage[7]);
	shuttleID ACCESS ADR(interface.Trak.Data[0]);
END_PROGRAM

PROGRAM _CYCLIC
	IF gSim = TRUE THEN
		bBlockReadOnceAck := bBlockReadOnce;
		bBlockSendOnceAck := bBlockSendOnce;
		bBlockSendShuttleIDAck := bBlockSendShuttleID;

		IF interface.Trak.ShuttleArrived = TRUE THEN
			interface.Equipment.Ready 		:= FALSE;

			tmr.IN 							:= TRUE;
			tmr.PT 							:= T#1s;
		END_IF

		IF tmr.Q = TRUE THEN
			interface.Equipment.Done 		:= TRUE;
		END_IF

		IF interface.Trak.ShuttleArrived = FALSE THEN
			tmr.IN							:= FALSE;
			interface.Equipment.Ready 		:= TRUE;
			interface.Equipment.Done 		:= FALSE;
		END_IF

		tmr();
	END_IF

	IF targetSlot.Interface = E_SLOT_UNKNOWN THEN
		step 				:= 0;
	END_IF

	CASE step OF
		0:	(* Modbus Interface Initialize and Shuttle Check *)
			bBlockSendShuttleID					:= FALSE;
			bBlockSendOnce						:= FALSE;
			bBlockReadOnce						:= FALSE;

			//interface.Trak.ShuttleArrived		:= FALSE;

			IF targetSlot.Shuttle.controlif <> 0 AND bBlockSendOnceAck = FALSE AND bBlockReadOnceAck = FALSE AND bBlockSendShuttleIDAck = FALSE THEN
				step 							:= 10;
			END_IF

		10:	(* Read Shuttle Data from userData *)
			fbUserData.DataAddress 				:= ADR(userData);
			fbUserData.DataSize 				:= SIZEOF(userData);
			fbUserData.Mode						:= mcACPTRAK_USERDATA_GET;
			fbUserData.Execute 					:= TRUE;

			IF fbUserData.Done = TRUE THEN
				//End to Read Data fron user Data
				fbUserData.Execute 				:= FALSE;

				//Copy User Data to Modbus IO
				brsmemcpy(ADR(interface.Trak.Data[0]),ADR(userData.SerialNumber), 11);
				brsmemcpy(ADR(interface.Trak.Data2[0]),ADR(userData.Data[0]), SIZEOF(userData.Data));

				//Start to Write userdata to Modbus
				bBlockSendOnce					:= TRUE;
				bBlockSendShuttleID				:= TRUE;
				step 							:= 11;
			END_IF

		11: (* Check End of write to Modbus *)
			IF bBlockSendOnceAck AND bBlockSendShuttleIDAck THEN
				bBlockSendOnce					:= FALSE;
				bBlockSendShuttleID				:= FALSE;
				step							:= 20;
			END_IF

		20: (* Check Process Ready *)
			IF targetSlot.Interface = E_SLOT_PROCESS_READY THEN
				step 							:= 30;
			ELSIF targetSlot.Shuttle.controlif = 0 THEN
				step 							:= 0;
			END_IF

		30:	(* Check Assemble Status and Slot Status *)
			IF (gSts.AsmState = E_ASM_PROCESS OR gSts.AsmState = E_ASM_IDLE)
				AND targetSlot.Interface = E_SLOT_PROCESS_READY THEN
				interface.Trak.ShuttleArrived	:= TRUE;
				fbShuttleOutCheck.Enable		:= TRUE;
				step 							:= 100;
			END_IF

		100: (* Wait Proess End and Next Stage Ready *)
			IF interface.Equipment.Done = TRUE AND NextReady THEN
				//Start to Read Data from PLC
				bBlockReadOnce					:= TRUE;
				step 							:= 101;
			END_IF

		101:
			IF bBlockReadOnceAck = TRUE THEN
				// Save Current Process Status
				userData.ProcessStatus			:= currentProcess;

				// Read process data from PLC
				brsmemcpy(ADR(userData.Data[0]), ADR(interface.Equipment.Data2[0]), SIZEOF(interface.Equipment.Data2));

				// End to Read Data from PLC
				bBlockReadOnce					:= FALSE;
				step := 110;
			END_IF

		110: 	//Write User Data
			fbUserData.DataAddress 				:= ADR(userData);
			fbUserData.DataSize 				:= SIZE_OF_USERDATA;
			fbUserData.Mode						:= mcACPTRAK_USERDATA_SET;
			fbUserData.Execute 					:= TRUE;

			IF fbUserData.Done = TRUE THEN
				fbUserData.Execute 				:= FALSE;
				//	interface.Trak.ShuttleArrived 	:= FALSE;
				targetSlot.Interface 			:= E_SLOT_TAKEOUT_READY;
				targetSlot.NextStage			:= nextSlot;
				step 							:= 120;
			END_IF

		120: 	//Done Check
			IF interface.Equipment.Done = FALSE THEN
				step 						:= 0;
			END_IF
	END_CASE;

	IF fbShuttleOutCheck.EventCount > 0 THEN
		interface.Trak.ShuttleArrived	:= FALSE;
		fbShuttleOutCheck.Enable		:= FALSE;
	END_IF

	IF targetSlot.Shuttle.controlif = 0 AND shuttleID <> '' THEN
		brsmemset(ADR(interface.Trak.Data[0]),0,11);
	END_IF

	fbUserData();
	fbShuttleOutCheck();
	Timer();
	Timer2();

END_PROGRAM
```

### Program Logical/Source/Control/ifStage9 (IEC) - CCR 2

#### Main.st
```iecst
PROGRAM _INIT
	currentProcess							:= E_PROCESS_Stage9;
	fbUserData.Axis							:= ADR(StStage[8].Shuttle);
	nextSlot 								:= ADR(StStage[9]);

	fbShuttleOutCheck.ProcessPoint			:= ADR(ptStage9);

	targetSlot ACCESS ADR(StStage[8]);
	shuttleID ACCESS ADR(interface.Trak.Data[0]);

	NextReady 								:= TRUE;
END_PROGRAM

PROGRAM _CYCLIC
	IF gSim = TRUE THEN
		bBlockReadOnceAck := bBlockReadOnce;
		bBlockSendOnceAck := bBlockSendOnce;
		bBlockSendShuttleIDAck := bBlockSendShuttleID;

		IF interface.Trak.ShuttleArrived = TRUE THEN
			interface.Equipment.Ready 		:= FALSE;

			tmr.IN 							:= TRUE;
			tmr.PT 							:= T#1s;
		END_IF

		IF tmr.Q = TRUE THEN
			interface.Equipment.Done 		:= TRUE;
		END_IF

		IF interface.Trak.ShuttleArrived = FALSE THEN
			tmr.IN							:= FALSE;
			interface.Equipment.Ready 		:= TRUE;
			interface.Equipment.Done 		:= FALSE;
		END_IF

		tmr();
	END_IF

	IF targetSlot.Interface = E_SLOT_UNKNOWN THEN
		step 				:= 0;
	END_IF

	CASE step OF
		0:	(* Modbus Interface Initialize and Shuttle Check *)
			bBlockSendShuttleID					:= FALSE;
			bBlockSendOnce						:= FALSE;
			bBlockReadOnce						:= FALSE;

			//interface.Trak.ShuttleArrived		:= FALSE;

			IF targetSlot.Shuttle.controlif <> 0 AND bBlockSendOnceAck = FALSE AND bBlockReadOnceAck = FALSE AND bBlockSendShuttleIDAck = FALSE THEN
				step 							:= 10;
			END_IF

		10:	(* Read Shuttle Data from userData *)
			fbUserData.DataAddress 				:= ADR(userData);
			fbUserData.DataSize 				:= SIZEOF(userData);
			fbUserData.Mode						:= mcACPTRAK_USERDATA_GET;
			fbUserData.Execute 					:= TRUE;

			IF fbUserData.Done = TRUE THEN
				//End to Read Data fron user Data
				fbUserData.Execute 				:= FALSE;

				//Copy User Data to Modbus IO
				brsmemcpy(ADR(interface.Trak.Data[0]),ADR(userData.SerialNumber), 11);
				brsmemcpy(ADR(interface.Trak.Data2[0]),ADR(userData.Data[0]), SIZEOF(userData.Data));

				//Start to Write userdata to Modbus
				bBlockSendOnce					:= TRUE;
				bBlockSendShuttleID				:= TRUE;
				step 							:= 11;
			END_IF

		11: (* Check End of write to Modbus *)
			IF bBlockSendOnceAck AND bBlockSendShuttleIDAck THEN
				bBlockSendOnce					:= FALSE;
				bBlockSendShuttleID				:= FALSE;
				step							:= 20;
			END_IF

		20: (* Check Process Ready *)
			IF targetSlot.Interface = E_SLOT_PROCESS_READY THEN
				step 							:= 30;
			ELSIF targetSlot.Shuttle.controlif = 0 THEN
				step 							:= 0;
			END_IF

		30:	(* Check Assemble Status and Slot Status *)
			IF (gSts.AsmState = E_ASM_PROCESS OR gSts.AsmState = E_ASM_IDLE)
				AND targetSlot.Interface = E_SLOT_PROCESS_READY THEN
				interface.Trak.ShuttleArrived	:= TRUE;
				fbShuttleOutCheck.Enable		:= TRUE;
				step 							:= 100;
			END_IF

		100: (* Wait Proess End and Next Stage Ready *)
			IF interface.Equipment.Done = TRUE AND NextReady THEN
				//Start to Read Data from PLC
				bBlockReadOnce					:= TRUE;
				step 							:= 101;
			END_IF

		101:
			IF bBlockReadOnceAck = TRUE THEN
				// Save Current Process Status
				userData.ProcessStatus			:= currentProcess;

				// Read process data from PLC
				brsmemcpy(ADR(userData.Data[0]), ADR(interface.Equipment.Data2[0]), SIZEOF(interface.Equipment.Data2));

				// End to Read Data from PLC
				bBlockReadOnce					:= FALSE;
				step := 110;
			END_IF

		110: 	//Write User Data
			fbUserData.DataAddress 				:= ADR(userData);
			fbUserData.DataSize 				:= SIZE_OF_USERDATA;
			fbUserData.Mode						:= mcACPTRAK_USERDATA_SET;
			fbUserData.Execute 					:= TRUE;

			IF fbUserData.Done = TRUE THEN
				fbUserData.Execute 				:= FALSE;
				//	interface.Trak.ShuttleArrived 	:= FALSE;
				targetSlot.Interface 			:= E_SLOT_TAKEOUT_READY;
				targetSlot.NextStage			:= nextSlot;
				step 							:= 120;
			END_IF

		120: 	//Done Check
			IF interface.Equipment.Done = FALSE THEN
				step 						:= 0;
			END_IF
	END_CASE;

	IF fbShuttleOutCheck.EventCount > 0 THEN
		interface.Trak.ShuttleArrived	:= FALSE;
		fbShuttleOutCheck.Enable		:= FALSE;
	END_IF

	IF targetSlot.Shuttle.controlif = 0 AND shuttleID <> '' THEN
		brsmemset(ADR(interface.Trak.Data[0]),0,11);
	END_IF

	fbUserData();
	fbShuttleOutCheck();
	Timer();
	Timer2();

END_PROGRAM
```

### Program Logical/Source/Control/ifStage10 (IEC) - Maint

#### Main.st
```iecst
PROGRAM _INIT
	currentProcess							:= E_PROCESS_Stage10;
	fbUserData.Axis							:= ADR(StStage[9].Shuttle);
	nextSlot 								:= ADR(StStage[10]);

	fbShuttleOutCheck.ProcessPoint			:= ADR(ptStage10);

	targetSlot ACCESS ADR(StStage[9]);
	shuttleID ACCESS ADR(interface.Trak.Data[0]);
END_PROGRAM

PROGRAM _CYCLIC
	IF gSim = TRUE THEN
		bBlockReadOnceAck := bBlockReadOnce;
		bBlockSendOnceAck := bBlockSendOnce;
		bBlockSendShuttleIDAck := bBlockSendShuttleID;

		IF interface.Trak.ShuttleArrived = TRUE THEN
			interface.Equipment.Ready 		:= FALSE;

			tmr.IN 							:= TRUE;
			tmr.PT 							:= T#1s;
		END_IF

		IF tmr.Q = TRUE THEN
			interface.Equipment.Done 		:= TRUE;
		END_IF

		IF interface.Trak.ShuttleArrived = FALSE THEN
			tmr.IN							:= FALSE;
			interface.Equipment.Ready 		:= TRUE;
			interface.Equipment.Done 		:= FALSE;
		END_IF

		tmr();
	END_IF

	IF targetSlot.Interface = E_SLOT_UNKNOWN THEN
		step 				:= 0;
	END_IF

	CASE step OF
		0:	(* Modbus Interface Initialize and Shuttle Check *)
			bBlockSendShuttleID					:= FALSE;
			bBlockSendOnce						:= FALSE;
			bBlockReadOnce						:= FALSE;

			//interface.Trak.ShuttleArrived		:= FALSE;

			IF targetSlot.Shuttle.controlif <> 0 AND bBlockSendOnceAck = FALSE AND bBlockReadOnceAck = FALSE AND bBlockSendShuttleIDAck = FALSE THEN
				step 							:= 10;
			END_IF

		10:	(* Read Shuttle Data from userData *)
			fbUserData.DataAddress 				:= ADR(userData);
			fbUserData.DataSize 				:= SIZEOF(userData);
			fbUserData.Mode						:= mcACPTRAK_USERDATA_GET;
			fbUserData.Execute 					:= TRUE;

			IF fbUserData.Done = TRUE THEN
				//End to Read Data fron user Data
				fbUserData.Execute 				:= FALSE;

				//Copy User Data to Modbus IO
				brsmemcpy(ADR(interface.Trak.Data[0]),ADR(userData.SerialNumber), 11);
				brsmemcpy(ADR(interface.Trak.Data2[0]),ADR(userData.Data[0]), SIZEOF(userData.Data));

				//Start to Write userdata to Modbus
				bBlockSendOnce					:= TRUE;
				bBlockSendShuttleID				:= TRUE;
				step 							:= 11;
			END_IF

		11: (* Check End of write to Modbus *)
			IF bBlockSendOnceAck AND bBlockSendShuttleIDAck THEN
				bBlockSendOnce					:= FALSE;
				bBlockSendShuttleID				:= FALSE;
				step							:= 20;
			END_IF

		20: (* Check Process Ready *)
			IF targetSlot.Interface = E_SLOT_PROCESS_READY THEN
				step 							:= 30;
			ELSIF targetSlot.Shuttle.controlif = 0 THEN
				step 							:= 0;
			END_IF

		30:	(* Check Assemble Status and Slot Status *)
			IF (gSts.AsmState = E_ASM_PROCESS OR gSts.AsmState = E_ASM_IDLE)
				AND targetSlot.Interface = E_SLOT_PROCESS_READY THEN
				interface.Trak.ShuttleArrived	:= TRUE;
				fbShuttleOutCheck.Enable		:= TRUE;
				step 							:= 100;
			END_IF

		100: (* Wait Proess End and Next Stage Ready *)
			IF interface.Equipment.Done = TRUE AND NextReady THEN
				//Start to Read Data from PLC
				bBlockReadOnce					:= TRUE;
				step 							:= 101;
			END_IF

		101:
			IF bBlockReadOnceAck = TRUE THEN
				// Save Current Process Status
				userData.ProcessStatus			:= currentProcess;

				// Read process data from PLC
				brsmemcpy(ADR(userData.Data[0]), ADR(interface.Equipment.Data2[0]), SIZEOF(interface.Equipment.Data2));

				// End to Read Data from PLC
				bBlockReadOnce					:= FALSE;
				step := 110;
			END_IF

		110: 	//Write User Data
			fbUserData.DataAddress 				:= ADR(userData);
			fbUserData.DataSize 				:= SIZE_OF_USERDATA;
			fbUserData.Mode						:= mcACPTRAK_USERDATA_SET;
			fbUserData.Execute 					:= TRUE;

			IF fbUserData.Done = TRUE THEN
				fbUserData.Execute 				:= FALSE;
				//	interface.Trak.ShuttleArrived 	:= FALSE;
				targetSlot.Interface 			:= E_SLOT_TAKEOUT_READY;
				targetSlot.NextStage			:= nextSlot;
				step 							:= 120;
			END_IF

		120: 	//Done Check
			IF interface.Equipment.Done = FALSE THEN
				step 						:= 0;
			END_IF
	END_CASE;

	IF fbShuttleOutCheck.EventCount > 0 THEN
		interface.Trak.ShuttleArrived	:= FALSE;
		fbShuttleOutCheck.Enable		:= FALSE;
	END_IF

	IF targetSlot.Shuttle.controlif = 0 AND shuttleID <> '' THEN
		brsmemset(ADR(interface.Trak.Data[0]),0,11);
	END_IF

	fbUserData();
	fbShuttleOutCheck();
	Timer();
	Timer2();

END_PROGRAM
```

### Program Logical/Source/Control/ifStage11 (IEC) - CCR 2 vision
